LIN {X 0,Y 514.541,Z 472.109,A -85,B 0,C 180,E1 18530.323,E2 18530.323} C_VEL
LIN {X 0,Y 518.512,Z 477.461,A -85,B 0,C 180,E1 18528.318,E2 18528.318} C_VEL
LIN {X 0,Y 522.762,Z 483.32,A -85,B 0,C 180,E1 18526.449,E2 18526.449} C_VEL
LIN {X 0,Y 527.071,Z 489.295,A -85,B 0,C 180,E1 18524.767,E2 18524.767} C_VEL
LIN {X 0,Y 533.694,Z 498.743,A -85,B 0,C 180,E1 18522.472,E2 18522.472} C_VEL
LIN {X 0,Y 539.059,Z 506.974,A -85,B 0,C 180,E1 18520.795,E2 18520.795} C_VEL
LIN {X 0,Y 523.952,Z 728.007,A -85,B 0,C 180,E1 18517.35,E2 18517.35} C_VEL
LIN {X 0,Y 517.723,Z 820.272,A -85,B 0,C 180,E1 18515.894,E2 18515.894} C_VEL
LIN {X 0,Y 514.589,Z 848.021,A -85,B 0,C 180,E1 18515.355,E2 18515.355} C_VEL
LIN {X 0,Y 510.56,Z 873.327,A -85,B 0,C 180,E1 18514.692,E2 18514.692} C_VEL
LIN {X 0,Y 506.518,Z 894.443,A -85,B 0,C 180,E1 18514.008,E2 18514.008} C_VEL
LIN {X 0,Y 502.104,Z 914.553,A -85,B 0,C 180,E1 18513.226,E2 18513.226} C_VEL
LIN {X 0,Y 497.165,Z 934.488,A -85,B 0,C 180,E1 18512.317,E2 18512.317} C_VEL
LIN {X 0,Y 491.161,Z 956.295,A -85,B 0,C 180,E1 18511.152,E2 18511.152} C_VEL
LIN {X 0,Y 483.255,Z 981.832,A -85,B 0,C 180,E1 18509.524,E2 18509.524} C_VEL
LIN {X 0,Y 476.642,Z 1001.338,A -85,B 0,C 180,E1 18508.063,E2 18508.063} C_VEL
LIN {X 0,Y 470.058,Z 1019.621,A -85,B 0,C 180,E1 18506.493,E2 18506.493} C_VEL
LIN {X 0,Y 462.853,Z 1038.675,A -85,B 0,C 180,E1 18504.623,E2 18504.623} C_VEL
LIN {X 0,Y 453.945,Z 1061.048,A -85,B 0,C 180,E1 18502.048,E2 18502.048} C_VEL
LIN {X 0,Y 447.24,Z 1077.33,A -85,B 0,C 180,E1 18499.87,E2 18499.87} C_VEL
LIN {X 0,Y 441.126,Z 1092.029,A -85,B 0,C 180,E1 18497.639,E2 18497.639} C_VEL
LIN {X 0,Y 434.952,Z 1106.936,A -85,B 0,C 180,E1 18495.074,E2 18495.074} C_VEL
LIN {X 0,Y 427.824,Z 1124.354,A -85,B 0,C 180,E1 18491.585,E2 18491.585} C_VEL
LIN {X 0,Y 423.062,Z 1136.506,A -85,B 0,C 180,E1 18488.744,E2 18488.744} C_VEL
LIN {X 0,Y 419.152,Z 1147.094,A -85,B 0,C 180,E1 18485.931,E2 18485.931} C_VEL
LIN {X 0,Y 415.76,Z 1157.018,A -85,B 0,C 180,E1 18482.922,E2 18482.922} C_VEL
LIN {X 0,Y 412.455,Z 1168.021,A -85,B 0,C 180,E1 18479.001,E2 18479.001} C_VEL
LIN {X 0,Y 410.434,Z 1175.985,A -85,B 0,C 180,E1 18475.543,E2 18475.543} C_VEL
LIN {X 0,Y 409.286,Z 1181.753,A -85,B 0,C 180,E1 18472.553,E2 18472.553} C_VEL
LIN {X 0,Y 408.55,Z 1186.458,A -85,B 0,C 180,E1 18469.59,E2 18469.59} C_VEL
LIN {X 0,Y 408.161,Z 1190.139,A -85,B 0,C 180,E1 18466.655,E2 18466.655} C_VEL
LIN {X 0,Y 407.98,Z 1192.833,A -85,B 0,C 180,E1 18463.752,E2 18463.752} C_VEL
LIN {X 0,Y 407.922,Z 1194.569,A -85,B 0,C 180,E1 18460.879,E2 18460.879} C_VEL
LIN {X 0,Y 407.905,Z 1195.381,A -85,B 0,C 180,E1 18457.977,E2 18457.977} C_VEL
LIN {X 0,Y 407.916,Z 1195.427,A -85,B 0,C 180,E1 18456.222,E2 18456.222} C_VEL
LIN {X 0,Y 406.93,Z 1195.271,A -85,B 0,C 180,E1 18455.141,E2 18455.141} C_VEL
LIN {X 0,Y 402.464,Z 1194.759,A -85,B 0,C 180,E1 18453.178,E2 18453.178} C_VEL
LIN {X 0,Y 400.134,Z 1194.102,A -85,B 0,C 180,E1 18451.777,E2 18451.777} C_VEL
LIN {X 0,Y 399.947,Z 1193.873,A -85,B 0,C 180,E1 18451.298,E2 18451.298} C_VEL
LIN {X 0,Y 400.135,Z 1190.746,A -85,B 0,C 180,E1 18447.565,E2 18447.565} C_VEL
LIN {X 0,Y 400.536,Z 1186.971,A -85,B 0,C 180,E1 18444.413,E2 18444.413} C_VEL
LIN {X 0,Y 401.262,Z 1182.348,A -85,B 0,C 180,E1 18441.402,E2 18441.402} C_VEL
LIN {X 0,Y 402.426,Z 1176.694,A -85,B 0,C 180,E1 18438.39,E2 18438.39} C_VEL
LIN {X 0,Y 404.11,Z 1169.973,A -85,B 0,C 180,E1 18435.382,E2 18435.382} C_VEL
LIN {X 0,Y 406.636,Z 1161.349,A -85,B 0,C 180,E1 18432.1,E2 18432.1} C_VEL
LIN {X 0,Y 410.803,Z 1148.852,A -85,B 0,C 180,E1 18428.137,E2 18428.137} C_VEL
LIN {X 0,Y 414.762,Z 1137.944,A -85,B 0,C 180,E1 18425.2,E2 18425.2} C_VEL
LIN {X 0,Y 418.993,Z 1126.868,A -85,B 0,C 180,E1 18422.577,E2 18422.577} C_VEL
LIN {X 0,Y 423.994,Z 1114.24,A -85,B 0,C 180,E1 18419.939,E2 18419.939} C_VEL
LIN {X 0,Y 430.697,Z 1097.792,A -85,B 0,C 180,E1 18416.938,E2 18416.938} C_VEL
LIN {X 0,Y 437.793,Z 1079.937,A -85,B 0,C 180,E1 18414.174,E2 18414.174} C_VEL
LIN {X 0,Y 443.949,Z 1064.334,A -85,B 0,C 180,E1 18412.059,E2 18412.059} C_VEL
LIN {X 0,Y 450.043,Z 1048.496,A -85,B 0,C 180,E1 18410.159,E2 18410.159} C_VEL
LIN {X 0,Y 456.669,Z 1030.666,A -85,B 0,C 180,E1 18408.272,E2 18408.272} C_VEL
LIN {X 0,Y 465.037,Z 1006.737,A -85,B 0,C 180,E1 18406.101,E2 18406.101} C_VEL
LIN {X 0,Y 471.267,Z 987.54,A -85,B 0,C 180,E1 18404.611,E2 18404.611} C_VEL
LIN {X 0,Y 476.948,Z 968.674,A -85,B 0,C 180,E1 18403.328,E2 18403.328} C_VEL
LIN {X 0,Y 482.604,Z 948.292,A -85,B 0,C 180,E1 18402.124,E2 18402.124} C_VEL
LIN {X 0,Y 488.772,Z 923.824,A -85,B 0,C 180,E1 18400.892,E2 18400.892} C_VEL
LIN {X 0,Y 494.214,Z 898.257,A -85,B 0,C 180,E1 18399.846,E2 18399.846} C_VEL
LIN {X 0,Y 498.2,Z 876.459,A -85,B 0,C 180,E1 18399.111,E2 18399.111} C_VEL
LIN {X 0,Y 501.467,Z 855.255,A -85,B 0,C 180,E1 18398.525,E2 18398.525} C_VEL
LIN {X 0,Y 504.339,Z 832.162,A -85,B 0,C 180,E1 18398.02,E2 18398.02} C_VEL
LIN {X 0,Y 507.084,Z 796.287,A -85,B 0,C 180,E1 18397.415,E2 18397.415} C_VEL
LIN {X 0,Y 520.447,Z 572.17,A -85,B 0,C 180,E1 18393.945,E2 18393.945} C_VEL
LIN {X 0,Y 524.409,Z 506.936,A -85,B 0,C 180,E1 18392.916,E2 18392.916} C_VEL
LIN {X 0,Y 515.302,Z 493.27,A -85,B 0,C 180,E1 18390.589,E2 18390.589} C_VEL
LIN {X 0,Y 506.344,Z 480.4,A -85,B 0,C 180,E1 18388.033,E2 18388.033} C_VEL
LIN {X 0,Y 498.92,Z 470.251,A -85,B 0,C 180,E1 18385.651,E2 18385.651} C_VEL
LIN {X 0,Y 494.57,Z 464.457,A -85,B 0,C 180,E1 18384.104,E2 18384.104} C_VEL
LIN {X 0,Y 491.363,Z 460.243,A -85,B 0,C 180,E1 18382.872,E2 18382.872} C_VEL
LIN {X 0,Y 487.688,Z 455.452,A -85,B 0,C 180,E1 18381.341,E2 18381.341} C_VEL
LIN {X 0,Y 483.606,Z 450.143,A -85,B 0,C 180,E1 18379.444,E2 18379.444} C_VEL
LIN {X 0,Y 479.486,Z 444.918,A -85,B 0,C 180,E1 18377.244,E2 18377.244} C_VEL
LIN {X 0,Y 476.311,Z 441.329,A -85,B 0,C 180,E1 18375.275,E2 18375.275} C_VEL
LIN {X 0,Y 475.115,Z 439.249,A -85,B 0,C 180,E1 18374.379,E2 18374.379} C_VEL
LIN {X 0,Y 472.029,Z 436.36,A -85,B 0,C 180,E1 18371.857,E2 18371.857} C_VEL
LIN {X 0,Y 470.403,Z 433.167,A -85,B 0,C 180,E1 18369.914,E2 18369.914} C_VEL
LIN {X 0,Y 467.781,Z 431.545,A -85,B 0,C 180,E1 18364.045,E2 18364.045} C_VEL
LIN {X 0,Y 468.554,Z 432.213,A -85,B 0,C 180,E1 18360,E2 18360} C_VEL
LIN {X 0,Y 470.689,Z 433.52,A -85,B 0,C 180,E1 18356.834,E2 18356.834} C_VEL
LIN {X 0,Y 472.775,Z 437.369,A -85,B 0,C 180,E1 18354.539,E2 18354.539} C_VEL
LIN {X 0,Y 475.407,Z 439.641,A -85,B 0,C 180,E1 18352.507,E2 18352.507} C_VEL
LIN {X 0,Y 478.181,Z 443.702,A -85,B 0,C 180,E1 18350.613,E2 18350.613} C_VEL
LIN {X 0,Y 480.232,Z 445.708,A -85,B 0,C 180,E1 18349.442,E2 18349.442} C_VEL
LIN {X 0,Y 483.756,Z 450.314,A -85,B 0,C 180,E1 18347.587,E2 18347.587} C_VEL
LIN {X 0,Y 489.426,Z 457.654,A -85,B 0,C 180,E1 18345.023,E2 18345.023} C_VEL
LIN {X 0,Y 493.652,Z 463.214,A -85,B 0,C 180,E1 18343.345,E2 18343.345} C_VEL
LIN {X 0,Y 498.77,Z 470.057,A -85,B 0,C 180,E1 18341.503,E2 18341.503} C_VEL
LIN {X 0,Y 505.342,Z 478.953,A -85,B 0,C 180,E1 18339.378,E2 18339.378} C_VEL
LIN {X 0,Y 511.266,Z 487.935,A -85,B 0,C 180,E1 18337.612,E2 18337.612} C_VEL
LIN {X 0,Y 520.655,Z 502.964,A -85,B 0,C 180,E1 18335.068,E2 18335.068} C_VEL
LIN {X 0,Y 524.429,Z 509.627,A -85,B 0,C 180,E1 18334.109,E2 18334.109} C_VEL
LIN {X 0,Y 511.272,Z 727.01,A -85,B 0,C 180,E1 18330.736,E2 18330.736} C_VEL
LIN {X 0,Y 505.302,Z 825.794,A -85,B 0,C 180,E1 18329.189,E2 18329.189} C_VEL
LIN {X 0,Y 502.366,Z 853.611,A -85,B 0,C 180,E1 18328.652,E2 18328.652} C_VEL
LIN {X 0,Y 498.441,Z 879.544,A -85,B 0,C 180,E1 18327.977,E2 18327.977} C_VEL
LIN {X 0,Y 494.631,Z 900.61,A -85,B 0,C 180,E1 18327.295,E2 18327.295} C_VEL
LIN {X 0,Y 490.381,Z 921.029,A -85,B 0,C 180,E1 18326.504,E2 18326.504} C_VEL
LIN {X 0,Y 485.26,Z 942.822,A -85,B 0,C 180,E1 18325.505,E2 18325.505} C_VEL
LIN {X 0,Y 478.136,Z 969.65,A -85,B 0,C 180,E1 18324.025,E2 18324.025} C_VEL
LIN {X 0,Y 472.04,Z 990.095,A -85,B 0,C 180,E1 18322.69,E2 18322.69} C_VEL
LIN {X 0,Y 466.19,Z 1008.36,A -85,B 0,C 180,E1 18321.323,E2 18321.323} C_VEL
LIN {X 0,Y 460.135,Z 1026.2,A -85,B 0,C 180,E1 18319.805,E2 18319.805} C_VEL
LIN {X 0,Y 453.465,Z 1044.906,A -85,B 0,C 180,E1 18317.993,E2 18317.993} C_VEL
LIN {X 0,Y 444.933,Z 1067.602,A -85,B 0,C 180,E1 18315.428,E2 18315.428} C_VEL
LIN {X 0,Y 438.299,Z 1084.613,A -85,B 0,C 180,E1 18313.186,E2 18313.186} C_VEL
LIN {X 0,Y 432.59,Z 1099.07,A -85,B 0,C 180,E1 18311.027,E2 18311.027} C_VEL
LIN {X 0,Y 426.774,Z 1113.76,A -85,B 0,C 180,E1 18308.549,E2 18308.549} C_VEL
LIN {X 0,Y 420.3,Z 1130.399,A -85,B 0,C 180,E1 18305.314,E2 18305.314} C_VEL
LIN {X 0,Y 415.223,Z 1143.634,A -85,B 0,C 180,E1 18302.302,E2 18302.302} C_VEL
LIN {X 0,Y 411.387,Z 1154.324,A -85,B 0,C 180,E1 18299.526,E2 18299.526} C_VEL
LIN {X 0,Y 408.025,Z 1164.334,A -85,B 0,C 180,E1 18296.561,E2 18296.561} C_VEL
LIN {X 0,Y 405.122,Z 1173.984,A -85,B 0,C 180,E1 18293.259,E2 18293.259} C_VEL
LIN {X 0,Y 402.652,Z 1183.587,A -85,B 0,C 180,E1 18289.285,E2 18289.285} C_VEL
LIN {X 0,Y 401.344,Z 1189.964,A -85,B 0,C 180,E1 18286.053,E2 18286.053} C_VEL
LIN {X 0,Y 400.584,Z 1194.712,A -85,B 0,C 180,E1 18283.128,E2 18283.128} C_VEL
LIN {X 0,Y 400.164,Z 1198.608,A -85,B 0,C 180,E1 18280.103,E2 18280.103} C_VEL
LIN {X 0,Y 399.99,Z 1201.293,A -85,B 0,C 180,E1 18277.324,E2 18277.324} C_VEL
LIN {X 0,Y 399.919,Z 1203.173,A -85,B 0,C 180,E1 18274.445,E2 18274.445} C_VEL
LIN {X 0,Y 399.91,Z 1204.11,A -85,B 0,C 180,E1 18271.719,E2 18271.719} C_VEL
LIN {X 0,Y 399.913,Z 1204.201,A -85,B 0,C 180,E1 18268.854,E2 18268.854} C_VEL
LIN {X 0,Y 399.916,Z 1203.377,A -85,B 0,C 180,E1 18265.986,E2 18265.986} C_VEL
LIN {X 0,Y 399.967,Z 1201.638,A -85,B 0,C 180,E1 18263.108,E2 18263.108} C_VEL
LIN {X 0,Y 400.134,Z 1198.975,A -85,B 0,C 180,E1 18260.217,E2 18260.217} C_VEL
LIN {X 0,Y 400.528,Z 1195.167,A -85,B 0,C 180,E1 18257.163,E2 18257.163} C_VEL
LIN {X 0,Y 401.256,Z 1190.564,A -85,B 0,C 180,E1 18254.24,E2 18254.24} C_VEL
LIN {X 0,Y 402.439,Z 1184.673,A -85,B 0,C 180,E1 18251.157,E2 18251.157} C_VEL
LIN {X 0,Y 404.211,Z 1177.671,A -85,B 0,C 180,E1 18248.068,E2 18248.068} C_VEL
LIN {X 0,Y 407.314,Z 1167.466,A -85,B 0,C 180,E1 18244.247,E2 18244.247} C_VEL
LIN {X 0,Y 411.361,Z 1155.632,A -85,B 0,C 180,E1 18240.595,E2 18240.595} C_VEL
LIN {X 0,Y 415.406,Z 1144.863,A -85,B 0,C 180,E1 18237.701,E2 18237.701} C_VEL
LIN {X 0,Y 420.273,Z 1132.771,A -85,B 0,C 180,E1 18234.849,E2 18234.849} C_VEL
LIN {X 0,Y 426.871,Z 1117.144,A -85,B 0,C 180,E1 18231.632,E2 18231.632} C_VEL
LIN {X 0,Y 434.143,Z 1099.904,A -85,B 0,C 180,E1 18228.626,E2 18228.626} C_VEL
LIN {X 0,Y 440.46,Z 1085.089,A -85,B 0,C 180,E1 18226.363,E2 18226.363} C_VEL
LIN {X 0,Y 447.076,Z 1069.432,A -85,B 0,C 180,E1 18224.25,E2 18224.25} C_VEL
LIN {X 0,Y 455.489,Z 1049.155,A -85,B 0,C 180,E1 18221.862,E2 18221.862} C_VEL
LIN {X 0,Y 463.944,Z 1027.412,A -85,B 0,C 180,E1 18219.702,E2 18219.702} C_VEL
LIN {X 0,Y 470.794,Z 1008.909,A -85,B 0,C 180,E1 18218.107,E2 18218.107} C_VEL
LIN {X 0,Y 477.681,Z 989.169,A -85,B 0,C 180,E1 18216.625,E2 18216.625} C_VEL
LIN {X 0,Y 485.495,Z 965.019,A -85,B 0,C 180,E1 18215.072,E2 18215.072} C_VEL
LIN {X 0,Y 492.199,Z 941.436,A -85,B 0,C 180,E1 18213.814,E2 18213.814} C_VEL
LIN {X 0,Y 497.27,Z 921.68,A -85,B 0,C 180,E1 18212.917,E2 18212.917} C_VEL
LIN {X 0,Y 501.906,Z 901.407,A -85,B 0,C 180,E1 18212.135,E2 18212.135} C_VEL
LIN {X 0,Y 506.047,Z 880.54,A -85,B 0,C 180,E1 18211.461,E2 18211.461} C_VEL
LIN {X 0,Y 509.796,Z 858.126,A -85,B 0,C 180,E1 18210.873,E2 18210.873} C_VEL
LIN {X 0,Y 513.507,Z 828.706,A -85,B 0,C 180,E1 18210.283,E2 18210.283} C_VEL
LIN {X 0,Y 517.306,Z 776.027,A -85,B 0,C 180,E1 18209.44,E2 18209.44} C_VEL
LIN {X 0,Y 532.526,Z 555.952,A -85,B 0,C 180,E1 18206.005,E2 18206.005} C_VEL
LIN {X 0,Y 535.526,Z 513.871,A -85,B 0,C 180,E1 18205.34,E2 18205.34} C_VEL
LIN {X 0,Y 530.021,Z 504.697,A -85,B 0,C 180,E1 18203.516,E2 18203.516} C_VEL
LIN {X 0,Y 523.348,Z 494.052,A -85,B 0,C 180,E1 18201.021,E2 18201.021} C_VEL
LIN {X 0,Y 518.979,Z 487.856,A -85,B 0,C 180,E1 18199.177,E2 18199.177} C_VEL
LIN {X 0,Y 515.666,Z 483.285,A -85,B 0,C 180,E1 18197.607,E2 18197.607} C_VEL
LIN {X 0,Y 512.04,Z 478.241,A -85,B 0,C 180,E1 18195.633,E2 18195.633} C_VEL
LIN {X 0,Y 508.794,Z 473.79,A -85,B 0,C 180,E1 18193.525,E2 18193.525} C_VEL
LIN {X 0,Y 504.983,Z 468.841,A -85,B 0,C 180,E1 18190.247,E2 18190.247} C_VEL
LIN {X 0,Y 504.344,Z 467.593,A -85,B 0,C 180,E1 18189.471,E2 18189.471} C_VEL
LIN {X 0,Y 501.757,Z 465.408,A -85,B 0,C 180,E1 18184.114,E2 18184.114} C_VEL
LIN {X 0,Y 502.105,Z 465.864,A -85,B 0,C 180,E1 18181.027,E2 18181.027} C_VEL
LIN {X 0,Y 504.615,Z 467.919,A -85,B 0,C 180,E1 18177.007,E2 18177.007} C_VEL
LIN {X 0,Y 507.047,Z 472.025,A -85,B 0,C 180,E1 18174.568,E2 18174.568} C_VEL
LIN {X 0,Y 508.847,Z 473.888,A -85,B 0,C 180,E1 18173.229,E2 18173.229} C_VEL
LIN {X 0,Y 512.1,Z 478.311,A -85,B 0,C 180,E1 18171.127,E2 18171.127} C_VEL
LIN {X 0,Y 517.051,Z 485.162,A -85,B 0,C 180,E1 18168.511,E2 18168.511} C_VEL
LIN {X 0,Y 521.242,Z 491.03,A -85,B 0,C 180,E1 18166.635,E2 18166.635} C_VEL
LIN {X 0,Y 526.846,Z 498.837,A -85,B 0,C 180,E1 18164.45,E2 18164.45} C_VEL
LIN {X 0,Y 533.524,Z 508.845,A -85,B 0,C 180,E1 18162.156,E2 18162.156} C_VEL
LIN {X 0,Y 535.563,Z 512.091,A -85,B 0,C 180,E1 18161.506,E2 18161.506} C_VEL
LIN {X 0,Y 520.129,Z 731.771,A -85,B 0,C 180,E1 18158.081,E2 18158.081} C_VEL
LIN {X 0,Y 513.954,Z 820.365,A -85,B 0,C 180,E1 18156.681,E2 18156.681} C_VEL
LIN {X 0,Y 510.733,Z 848.221,A -85,B 0,C 180,E1 18156.141,E2 18156.141} C_VEL
LIN {X 0,Y 506.612,Z 873.503,A -85,B 0,C 180,E1 18155.482,E2 18155.482} C_VEL
LIN {X 0,Y 502.423,Z 894.86,A -85,B 0,C 180,E1 18154.793,E2 18154.793} C_VEL
LIN {X 0,Y 497.816,Z 915.254,A -85,B 0,C 180,E1 18154,E2 18154} C_VEL
LIN {X 0,Y 492.459,Z 936.22,A -85,B 0,C 180,E1 18153.039,E2 18153.039} C_VEL
LIN {X 0,Y 485.143,Z 961.704,A -85,B 0,C 180,E1 18151.645,E2 18151.645} C_VEL
LIN {X 0,Y 478.062,Z 983.47,A -85,B 0,C 180,E1 18150.223,E2 18150.223} C_VEL
LIN {X 0,Y 471.582,Z 1001.971,A -85,B 0,C 180,E1 18148.827,E2 18148.827} C_VEL
LIN {X 0,Y 464.808,Z 1020.203,A -85,B 0,C 180,E1 18147.255,E2 18147.255} C_VEL
LIN {X 0,Y 457.273,Z 1039.458,A -85,B 0,C 180,E1 18145.352,E2 18145.352} C_VEL
LIN {X 0,Y 448.172,Z 1061.456,A -85,B 0,C 180,E1 18142.799,E2 18142.799} C_VEL
LIN {X 0,Y 441.208,Z 1077.72,A -85,B 0,C 180,E1 18140.603,E2 18140.603} C_VEL
LIN {X 0,Y 434.858,Z 1092.389,A -85,B 0,C 180,E1 18138.354,E2 18138.354} C_VEL
LIN {X 0,Y 428.096,Z 1108.054,A -85,B 0,C 180,E1 18135.618,E2 18135.618} C_VEL
LIN {X 0,Y 420.991,Z 1124.623,A -85,B 0,C 180,E1 18132.231,E2 18132.231} C_VEL
LIN {X 0,Y 416.03,Z 1136.639,A -85,B 0,C 180,E1 18129.381,E2 18129.381} C_VEL
LIN {X 0,Y 411.869,Z 1147.312,A -85,B 0,C 180,E1 18126.496,E2 18126.496} C_VEL
LIN {X 0,Y 408.214,Z 1157.454,A -85,B 0,C 180,E1 18123.357,E2 18123.357} C_VEL
LIN {X 0,Y 404.669,Z 1168.563,A -85,B 0,C 180,E1 18119.281,E2 18119.281} C_VEL
LIN {X 0,Y 402.627,Z 1176.129,A -85,B 0,C 180,E1 18115.917,E2 18115.917} C_VEL
LIN {X 0,Y 401.384,Z 1181.959,A -85,B 0,C 180,E1 18112.822,E2 18112.822} C_VEL
LIN {X 0,Y 400.592,Z 1186.665,A -85,B 0,C 180,E1 18109.778,E2 18109.778} C_VEL
LIN {X 0,Y 400.17,Z 1190.408,A -85,B 0,C 180,E1 18106.699,E2 18106.699} C_VEL
LIN {X 0,Y 399.972,Z 1193.25,A -85,B 0,C 180,E1 18103.476,E2 18103.476} C_VEL
LIN {X 0,Y 399.919,Z 1195.192,A -85,B 0,C 180,E1 18099.788,E2 18099.788} C_VEL
LIN {X 0,Y 399.917,Z 1195.507,A -85,B 0,C 180,E1 18096.172,E2 18096.172} C_VEL
LIN {X 0,Y 399.921,Z 1194.742,A -85,B 0,C 180,E1 18093.153,E2 18093.153} C_VEL
LIN {X 0,Y 399.947,Z 1193.873,A -85,B 0,C 180,E1 18091.298,E2 18091.298} C_VEL
LIN {X 0,Y 398.997,Z 1193.239,A -85,B 0,C 180,E1 18090.198,E2 18090.198} C_VEL
LIN {X 0,Y 392.716,Z 1190.512,A -85,B 0,C 180,E1 18087.106,E2 18087.106} C_VEL
LIN {X 0,Y 392.26,Z 1189.666,A -85,B 0,C 180,E1 18086.302,E2 18086.302} C_VEL
LIN {X 0,Y 392.921,Z 1185.006,A -85,B 0,C 180,E1 18082.69,E2 18082.69} C_VEL
LIN {X 0,Y 394.336,Z 1177.904,A -85,B 0,C 180,E1 18078.593,E2 18078.593} C_VEL
LIN {X 0,Y 396.111,Z 1171.018,A -85,B 0,C 180,E1 18075.379,E2 18075.379} C_VEL
LIN {X 0,Y 398.426,Z 1163.313,A -85,B 0,C 180,E1 18072.323,E2 18072.323} C_VEL
LIN {X 0,Y 401.433,Z 1154.436,A -85,B 0,C 180,E1 18069.287,E2 18069.287} C_VEL
LIN {X 0,Y 406.061,Z 1142.105,A -85,B 0,C 180,E1 18065.657,E2 18065.657} C_VEL
LIN {X 0,Y 411.325,Z 1128.633,A -85,B 0,C 180,E1 18062.336,E2 18062.336} C_VEL
LIN {X 0,Y 416.314,Z 1116.454,A -85,B 0,C 180,E1 18059.712,E2 18059.712} C_VEL
LIN {X 0,Y 421.667,Z 1103.641,A -85,B 0,C 180,E1 18057.273,E2 18057.273} C_VEL
LIN {X 0,Y 427.606,Z 1089.446,A -85,B 0,C 180,E1 18054.886,E2 18054.886} C_VEL
LIN {X 0,Y 435.503,Z 1070.486,A -85,B 0,C 180,E1 18052.11,E2 18052.11} C_VEL
LIN {X 0,Y 442.917,Z 1051.844,A -85,B 0,C 180,E1 18049.788,E2 18049.788} C_VEL
LIN {X 0,Y 449.374,Z 1035.064,A -85,B 0,C 180,E1 18047.954,E2 18047.954} C_VEL
LIN {X 0,Y 455.747,Z 1017.743,A -85,B 0,C 180,E1 18046.285,E2 18046.285} C_VEL
LIN {X 0,Y 462.6,Z 998.079,A -85,B 0,C 180,E1 18044.626,E2 18044.626} C_VEL
LIN {X 0,Y 470.773,Z 972.483,A -85,B 0,C 180,E1 18042.795,E2 18042.795} C_VEL
LIN {X 0,Y 476.812,Z 951.552,A -85,B 0,C 180,E1 18041.53,E2 18041.53} C_VEL
LIN {X 0,Y 481.99,Z 931.83,A -85,B 0,C 180,E1 18040.502,E2 18040.502} C_VEL
LIN {X 0,Y 486.964,Z 910.669,A -85,B 0,C 180,E1 18039.557,E2 18039.557} C_VEL
LIN {X 0,Y 492.453,Z 883.629,A -85,B 0,C 180,E1 18038.561,E2 18038.561} C_VEL
LIN {X 0,Y 496.502,Z 858.808,A -85,B 0,C 180,E1 18037.846,E2 18037.846} C_VEL
LIN {X 0,Y 499.366,Z 837.111,A -85,B 0,C 180,E1 18037.352,E2 18037.352} C_VEL
LIN {X 0,Y 501.535,Z 814.579,A -85,B 0,C 180,E1 18036.942,E2 18036.942} C_VEL
LIN {X 0,Y 514.745,Z 600.28,A -85,B 0,C 180,E1 18033.606,E2 18033.606} C_VEL
LIN {X 0,Y 520.293,Z 511.555,A -85,B 0,C 180,E1 18032.21,E2 18032.21} C_VEL
LIN {X 0,Y 510.446,Z 496.68,A -85,B 0,C 180,E1 18029.58,E2 18029.58} C_VEL
LIN {X 0,Y 501.167,Z 483.294,A -85,B 0,C 180,E1 18026.769,E2 18026.769} C_VEL
LIN {X 0,Y 493.611,Z 472.979,A -85,B 0,C 180,E1 18024.154,E2 18024.154} C_VEL
LIN {X 0,Y 489.413,Z 467.465,A -85,B 0,C 180,E1 18022.524,E2 18022.524} C_VEL
LIN {X 0,Y 486.073,Z 463.017,A -85,B 0,C 180,E1 18021.1,E2 18021.1} C_VEL
LIN {X 0,Y 482.054,Z 457.73,A -85,B 0,C 180,E1 18019.194,E2 18019.194} C_VEL
LIN {X 0,Y 478.292,Z 452.785,A -85,B 0,C 180,E1 18017.144,E2 18017.144} C_VEL
LIN {X 0,Y 474.998,Z 449.034,A -85,B 0,C 180,E1 18015.069,E2 18015.069} C_VEL
LIN {X 0,Y 473.819,Z 447.031,A -85,B 0,C 180,E1 18014.17,E2 18014.17} C_VEL
LIN {X 0,Y 470.817,Z 444.076,A -85,B 0,C 180,E1 18011.64,E2 18011.64} C_VEL
LIN {X 0,Y 469.334,Z 441.079,A -85,B 0,C 180,E1 18009.813,E2 18009.813} C_VEL
LIN {X 0,Y 466.805,Z 439.485,A -85,B 0,C 180,E1 18004.053,E2 18004.053} C_VEL
LIN {X 0,Y 467.576,Z 440.157,A -85,B 0,C 180,E1 18000,E2 18000} C_VEL
LIN {X 0,Y 469.601,Z 441.436,A -85,B 0,C 180,E1 17996.949,E2 17996.949} C_VEL
LIN {X 0,Y 471.656,Z 445.241,A -85,B 0,C 180,E1 17994.648,E2 17994.648} C_VEL
LIN {X 0,Y 474.169,Z 447.478,A -85,B 0,C 180,E1 17992.67,E2 17992.67} C_VEL
LIN {X 0,Y 477.003,Z 451.586,A -85,B 0,C 180,E1 17990.711,E2 17990.711} C_VEL
LIN {X 0,Y 478.824,Z 453.407,A -85,B 0,C 180,E1 17989.654,E2 17989.654} C_VEL
LIN {X 0,Y 482.414,Z 458.106,A -85,B 0,C 180,E1 17987.734,E2 17987.734} C_VEL
LIN {X 0,Y 487.885,Z 465.381,A -85,B 0,C 180,E1 17985.217,E2 17985.217} C_VEL
LIN {X 0,Y 491.989,Z 470.863,A -85,B 0,C 180,E1 17983.56,E2 17983.56} C_VEL
LIN {X 0,Y 498.576,Z 479.657,A -85,B 0,C 180,E1 17981.193,E2 17981.193} C_VEL
LIN {X 0,Y 505.797,Z 489.962,A -85,B 0,C 180,E1 17978.882,E2 17978.882} C_VEL
LIN {X 0,Y 516.299,Z 506.899,A -85,B 0,C 180,E1 17975.881,E2 17975.881} C_VEL
LIN {X 0,Y 520.334,Z 513.973,A -85,B 0,C 180,E1 17974.816,E2 17974.816} C_VEL
LIN {X 0,Y 506.749,Z 732.106,A -85,B 0,C 180,E1 17971.427,E2 17971.427} C_VEL
LIN {X 0,Y 500.917,Z 825.772,A -85,B 0,C 180,E1 17969.955,E2 17969.955} C_VEL
LIN {X 0,Y 497.915,Z 853.564,A -85,B 0,C 180,E1 17969.418,E2 17969.418} C_VEL
LIN {X 0,Y 493.894,Z 879.509,A -85,B 0,C 180,E1 17968.745,E2 17968.745} C_VEL
LIN {X 0,Y 489.912,Z 900.999,A -85,B 0,C 180,E1 17968.049,E2 17968.049} C_VEL
LIN {X 0,Y 485.428,Z 921.952,A -85,B 0,C 180,E1 17967.234,E2 17967.234} C_VEL
LIN {X 0,Y 479.761,Z 945.371,A -85,B 0,C 180,E1 17966.15,E2 17966.15} C_VEL
LIN {X 0,Y 472.742,Z 970.746,A -85,B 0,C 180,E1 17964.725,E2 17964.725} C_VEL
LIN {X 0,Y 466.758,Z 990.243,A -85,B 0,C 180,E1 17963.446,E2 17963.446} C_VEL
LIN {X 0,Y 460.495,Z 1009.248,A -85,B 0,C 180,E1 17962.015,E2 17962.015} C_VEL
LIN {X 0,Y 454.024,Z 1027.724,A -85,B 0,C 180,E1 17960.423,E2 17960.423} C_VEL
LIN {X 0,Y 445.921,Z 1049.671,A -85,B 0,C 180,E1 17958.243,E2 17958.243} C_VEL
LIN {X 0,Y 438.21,Z 1069.244,A -85,B 0,C 180,E1 17955.95,E2 17955.95} C_VEL
LIN {X 0,Y 431.785,Z 1085.159,A -85,B 0,C 180,E1 17953.818,E2 17953.818} C_VEL
LIN {X 0,Y 425.54,Z 1100.435,A -85,B 0,C 180,E1 17951.498,E2 17951.498} C_VEL
LIN {X 0,Y 418.65,Z 1117.355,A -85,B 0,C 180,E1 17948.561,E2 17948.561} C_VEL
LIN {X 0,Y 412.34,Z 1132.708,A -85,B 0,C 180,E1 17945.418,E2 17945.418} C_VEL
LIN {X 0,Y 407.673,Z 1144.503,A -85,B 0,C 180,E1 17942.654,E2 17942.654} C_VEL
LIN {X 0,Y 403.742,Z 1155.023,A -85,B 0,C 180,E1 17939.853,E2 17939.853} C_VEL
LIN {X 0,Y 400.163,Z 1165.286,A -85,B 0,C 180,E1 17936.728,E2 17936.728} C_VEL
LIN {X 0,Y 396.693,Z 1176.5,A -85,B 0,C 180,E1 17932.683,E2 17932.683} C_VEL
LIN {X 0,Y 394.693,Z 1184.054,A -85,B 0,C 180,E1 17929.381,E2 17929.381} C_VEL
LIN {X 0,Y 393.4,Z 1190.089,A -85,B 0,C 180,E1 17926.235,E2 17926.235} C_VEL
LIN {X 0,Y 392.608,Z 1194.802,A -85,B 0,C 180,E1 17923.25,E2 17923.25} C_VEL
LIN {X 0,Y 392.174,Z 1198.605,A -85,B 0,C 180,E1 17920.214,E2 17920.214} C_VEL
LIN {X 0,Y 391.989,Z 1201.307,A -85,B 0,C 180,E1 17917.327,E2 17917.327} C_VEL
LIN {X 0,Y 391.92,Z 1203.078,A -85,B 0,C 180,E1 17914.536,E2 17914.536} C_VEL
LIN {X 0,Y 391.91,Z 1204.02,A -85,B 0,C 180,E1 17911.754,E2 17911.754} C_VEL
LIN {X 0,Y 391.914,Z 1204.115,A -85,B 0,C 180,E1 17908.831,E2 17908.831} C_VEL
LIN {X 0,Y 391.916,Z 1203.296,A -85,B 0,C 180,E1 17905.904,E2 17905.904} C_VEL
LIN {X 0,Y 391.976,Z 1201.5,A -85,B 0,C 180,E1 17902.887,E2 17902.887} C_VEL
LIN {X 0,Y 392.167,Z 1198.746,A -85,B 0,C 180,E1 17899.868,E2 17899.868} C_VEL
LIN {X 0,Y 392.579,Z 1195.11,A -85,B 0,C 180,E1 17896.899,E2 17896.899} C_VEL
LIN {X 0,Y 393.361,Z 1190.517,A -85,B 0,C 180,E1 17893.914,E2 17893.914} C_VEL
LIN {X 0,Y 394.633,Z 1184.643,A -85,B 0,C 180,E1 17890.769,E2 17890.769} C_VEL
LIN {X 0,Y 396.521,Z 1177.657,A -85,B 0,C 180,E1 17887.619,E2 17887.619} C_VEL
LIN {X 0,Y 399.807,Z 1167.483,A -85,B 0,C 180,E1 17883.727,E2 17883.727} C_VEL
LIN {X 0,Y 404.078,Z 1155.665,A -85,B 0,C 180,E1 17880.006,E2 17880.006} C_VEL
LIN {X 0,Y 408.343,Z 1144.933,A -85,B 0,C 180,E1 17877.072,E2 17877.072} C_VEL
LIN {X 0,Y 413.176,Z 1133.5,A -85,B 0,C 180,E1 17874.324,E2 17874.324} C_VEL
LIN {X 0,Y 419.791,Z 1118.462,A -85,B 0,C 180,E1 17871.158,E2 17871.158} C_VEL
LIN {X 0,Y 427.549,Z 1100.922,A -85,B 0,C 180,E1 17868.023,E2 17868.023} C_VEL
LIN {X 0,Y 434.479,Z 1085.311,A -85,B 0,C 180,E1 17865.606,E2 17865.606} C_VEL
LIN {X 0,Y 441.409,Z 1069.516,A -85,B 0,C 180,E1 17863.458,E2 17863.458} C_VEL
LIN {X 0,Y 450.068,Z 1049.385,A -85,B 0,C 180,E1 17861.074,E2 17861.074} C_VEL
LIN {X 0,Y 458.765,Z 1027.793,A -85,B 0,C 180,E1 17858.916,E2 17858.916} C_VEL
LIN {X 0,Y 465.815,Z 1009.353,A -85,B 0,C 180,E1 17857.32,E2 17857.32} C_VEL
LIN {X 0,Y 472.754,Z 990.059,A -85,B 0,C 180,E1 17855.864,E2 17855.864} C_VEL
LIN {X 0,Y 480.094,Z 968.131,A -85,B 0,C 180,E1 17854.44,E2 17854.44} C_VEL
LIN {X 0,Y 487.792,Z 942.188,A -85,B 0,C 180,E1 17853.034,E2 17853.034} C_VEL
LIN {X 0,Y 493.396,Z 920.871,A -85,B 0,C 180,E1 17852.07,E2 17852.07} C_VEL
LIN {X 0,Y 498.158,Z 900.449,A -85,B 0,C 180,E1 17851.293,E2 17851.293} C_VEL
LIN {X 0,Y 502.445,Z 879.192,A -85,B 0,C 180,E1 17850.616,E2 17850.616} C_VEL
LIN {X 0,Y 506.831,Z 853.258,A -85,B 0,C 180,E1 17849.958,E2 17849.958} C_VEL
LIN {X 0,Y 510.116,Z 825.477,A -85,B 0,C 180,E1 17849.429,E2 17849.429} C_VEL
LIN {X 0,Y 517.254,Z 725.256,A -85,B 0,C 180,E1 17847.847,E2 17847.847} C_VEL
LIN {X 0,Y 532.153,Z 518.787,A -85,B 0,C 180,E1 17844.624,E2 17844.624} C_VEL
LIN {X 0,Y 524.714,Z 506.488,A -85,B 0,C 180,E1 17841.99,E2 17841.99} C_VEL
LIN {X 0,Y 520.347,Z 499.65,A -85,B 0,C 180,E1 17840.236,E2 17840.236} C_VEL
LIN {X 0,Y 516.932,Z 494.804,A -85,B 0,C 180,E1 17838.729,E2 17838.729} C_VEL
LIN {X 0,Y 514.042,Z 490.737,A -85,B 0,C 180,E1 17837.314,E2 17837.314} C_VEL
LIN {X 0,Y 510.694,Z 485.955,A -85,B 0,C 180,E1 17835.443,E2 17835.443} C_VEL
LIN {X 0,Y 507.513,Z 481.496,A -85,B 0,C 180,E1 17833.327,E2 17833.327} C_VEL
LIN {X 0,Y 503.822,Z 476.579,A -85,B 0,C 180,E1 17830.058,E2 17830.058} C_VEL
LIN {X 0,Y 503.275,Z 475.497,A -85,B 0,C 180,E1 17829.376,E2 17829.376} C_VEL
LIN {X 0,Y 500.771,Z 473.331,A -85,B 0,C 180,E1 17824.007,E2 17824.007} C_VEL
LIN {X 0,Y 501.163,Z 473.862,A -85,B 0,C 180,E1 17820.915,E2 17820.915} C_VEL
LIN {X 0,Y 503.499,Z 475.749,A -85,B 0,C 180,E1 17817.154,E2 17817.154} C_VEL
LIN {X 0,Y 506.062,Z 480.048,A -85,B 0,C 180,E1 17814.558,E2 17814.558} C_VEL
LIN {X 0,Y 507.621,Z 481.704,A -85,B 0,C 180,E1 17813.383,E2 17813.383} C_VEL
LIN {X 0,Y 510.922,Z 486.191,A -85,B 0,C 180,E1 17811.22,E2 17811.22} C_VEL
LIN {X 0,Y 515.597,Z 492.859,A -85,B 0,C 180,E1 17808.704,E2 17808.704} C_VEL
LIN {X 0,Y 519.604,Z 498.553,A -85,B 0,C 180,E1 17806.875,E2 17806.875} C_VEL
LIN {X 0,Y 524.981,Z 506.177,A -85,B 0,C 180,E1 17804.733,E2 17804.733} C_VEL
LIN {X 0,Y 531.55,Z 516.198,A -85,B 0,C 180,E1 17802.427,E2 17802.427} C_VEL
LIN {X 0,Y 532.146,Z 517.318,A -85,B 0,C 180,E1 17802.225,E2 17802.225} C_VEL
LIN {X 0,Y 516.403,Z 735.346,A -85,B 0,C 180,E1 17798.826,E2 17798.826} C_VEL
LIN {X 0,Y 510.276,Z 820.692,A -85,B 0,C 180,E1 17797.476,E2 17797.476} C_VEL
LIN {X 0,Y 506.932,Z 848.728,A -85,B 0,C 180,E1 17796.933,E2 17796.933} C_VEL
LIN {X 0,Y 502.763,Z 873.691,A -85,B 0,C 180,E1 17796.285,E2 17796.285} C_VEL
LIN {X 0,Y 498.633,Z 894.312,A -85,B 0,C 180,E1 17795.624,E2 17795.624} C_VEL
LIN {X 0,Y 493.842,Z 915.065,A -85,B 0,C 180,E1 17794.826,E2 17794.826} C_VEL
LIN {X 0,Y 488.471,Z 935.626,A -85,B 0,C 180,E1 17793.89,E2 17793.89} C_VEL
LIN {X 0,Y 481.459,Z 959.677,A -85,B 0,C 180,E1 17792.598,E2 17792.598} C_VEL
LIN {X 0,Y 473.589,Z 983.262,A -85,B 0,C 180,E1 17791.07,E2 17791.07} C_VEL
LIN {X 0,Y 466.701,Z 1002.388,A -85,B 0,C 180,E1 17789.627,E2 17789.627} C_VEL
LIN {X 0,Y 459.644,Z 1020.788,A -85,B 0,C 180,E1 17788.034,E2 17788.034} C_VEL
LIN {X 0,Y 451.254,Z 1041.555,A -85,B 0,C 180,E1 17785.963,E2 17785.963} C_VEL
LIN {X 0,Y 442.317,Z 1062.237,A -85,B 0,C 180,E1 17783.521,E2 17783.521} C_VEL
LIN {X 0,Y 435.258,Z 1078.127,A -85,B 0,C 180,E1 17781.355,E2 17781.355} C_VEL
LIN {X 0,Y 428.496,Z 1093.135,A -85,B 0,C 180,E1 17779.026,E2 17779.026} C_VEL
LIN {X 0,Y 420.947,Z 1109.985,A -85,B 0,C 180,E1 17776.03,E2 17776.03} C_VEL
LIN {X 0,Y 413.91,Z 1125.575,A -85,B 0,C 180,E1 17772.745,E2 17772.745} C_VEL
LIN {X 0,Y 408.756,Z 1137.483,A -85,B 0,C 180,E1 17769.857,E2 17769.857} C_VEL
LIN {X 0,Y 404.422,Z 1148.073,A -85,B 0,C 180,E1 17766.925,E2 17766.925} C_VEL
LIN {X 0,Y 399.992,Z 1159.927,A -85,B 0,C 180,E1 17763.13,E2 17763.13} C_VEL
LIN {X 0,Y 396.683,Z 1169.767,A -85,B 0,C 180,E1 17759.291,E2 17759.291} C_VEL
LIN {X 0,Y 394.758,Z 1176.594,A -85,B 0,C 180,E1 17756.149,E2 17756.149} C_VEL
LIN {X 0,Y 393.466,Z 1182.282,A -85,B 0,C 180,E1 17753.038,E2 17753.038} C_VEL
LIN {X 0,Y 392.631,Z 1186.911,A -85,B 0,C 180,E1 17749.952,E2 17749.952} C_VEL
LIN {X 0,Y 392.18,Z 1190.684,A -85,B 0,C 180,E1 17746.744,E2 17746.744} C_VEL
LIN {X 0,Y 391.964,Z 1193.724,A -85,B 0,C 180,E1 17743.122,E2 17743.122} C_VEL
LIN {X 0,Y 391.916,Z 1195.35,A -85,B 0,C 180,E1 17739.397,E2 17739.397} C_VEL
LIN {X 0,Y 391.917,Z 1195.592,A -85,B 0,C 180,E1 17736.151,E2 17736.151} C_VEL
LIN {X 0,Y 391.923,Z 1194.82,A -85,B 0,C 180,E1 17733.071,E2 17733.071} C_VEL
LIN {X 0,Y 391.996,Z 1193.069,A -85,B 0,C 180,E1 17730,E2 17730} C_VEL
LIN {X 0,Y 392.196,Z 1190.339,A -85,B 0,C 180,E1 17726.931,E2 17726.931} C_VEL
LIN {X 0,Y 392.26,Z 1189.666,A -85,B 0,C 180,E1 17726.302,E2 17726.302} C_VEL
LIN {X 0,Y 391.408,Z 1188.503,A -85,B 0,C 180,E1 17725.188,E2 17725.188} C_VEL
LIN {X 0,Y 385.611,Z 1184.551,A -85,B 0,C 180,E1 17722.048,E2 17722.048} C_VEL
LIN {X 0,Y 385.324,Z 1183.25,A -85,B 0,C 180,E1 17721.242,E2 17721.242} C_VEL
LIN {X 0,Y 386.667,Z 1177.336,A -85,B 0,C 180,E1 17717.91,E2 17717.91} C_VEL
LIN {X 0,Y 388.518,Z 1170.68,A -85,B 0,C 180,E1 17714.782,E2 17714.782} C_VEL
LIN {X 0,Y 390.997,Z 1162.909,A -85,B 0,C 180,E1 17711.667,E2 17711.667} C_VEL
LIN {X 0,Y 394.535,Z 1153.069,A -85,B 0,C 180,E1 17708.284,E2 17708.284} C_VEL
LIN {X 0,Y 399.872,Z 1139.485,A -85,B 0,C 180,E1 17704.369,E2 17704.369} C_VEL
LIN {X 0,Y 404.672,Z 1127.923,A -85,B 0,C 180,E1 17701.52,E2 17701.52} C_VEL
LIN {X 0,Y 409.935,Z 1115.658,A -85,B 0,C 180,E1 17698.863,E2 17698.863} C_VEL
LIN {X 0,Y 415.882,Z 1101.998,A -85,B 0,C 180,E1 17696.264,E2 17696.264} C_VEL
LIN {X 0,Y 423.606,Z 1084.277,A -85,B 0,C 180,E1 17693.333,E2 17693.333} C_VEL
LIN {X 0,Y 431.162,Z 1066.313,A -85,B 0,C 180,E1 17690.808,E2 17690.808} C_VEL
LIN {X 0,Y 437.894,Z 1049.945,A -85,B 0,C 180,E1 17688.796,E2 17688.796} C_VEL
LIN {X 0,Y 444.388,Z 1033.556,A -85,B 0,C 180,E1 17687.02,E2 17687.02} C_VEL
LIN {X 0,Y 451.484,Z 1014.764,A -85,B 0,C 180,E1 17685.232,E2 17685.232} C_VEL
LIN {X 0,Y 459.98,Z 990.555,A -85,B 0,C 180,E1 17683.266,E2 17683.266} C_VEL
LIN {X 0,Y 466.496,Z 970.165,A -85,B 0,C 180,E1 17681.858,E2 17681.858} C_VEL
LIN {X 0,Y 472.16,Z 950.889,A -85,B 0,C 180,E1 17680.702,E2 17680.702} C_VEL
LIN {X 0,Y 477.449,Z 931.176,A -85,B 0,C 180,E1 17679.682,E2 17679.682} C_VEL
LIN {X 0,Y 482.711,Z 909.23,A -85,B 0,C 180,E1 17678.711,E2 17678.711} C_VEL
LIN {X 0,Y 488.485,Z 880.723,A -85,B 0,C 180,E1 17677.687,E2 17677.687} C_VEL
LIN {X 0,Y 492.233,Z 858.042,A -85,B 0,C 180,E1 17677.045,E2 17677.045} C_VEL
LIN {X 0,Y 495.121,Z 836.463,A -85,B 0,C 180,E1 17676.559,E2 17676.559} C_VEL
LIN {X 0,Y 497.365,Z 813.232,A -85,B 0,C 180,E1 17676.14,E2 17676.14} C_VEL
LIN {X 0,Y 511.116,Z 596.254,A -85,B 0,C 180,E1 17672.759,E2 17672.759} C_VEL
LIN {X 0,Y 516.277,Z 516.161,A -85,B 0,C 180,E1 17671.496,E2 17671.496} C_VEL
LIN {X 0,Y 506.18,Z 500.884,A -85,B 0,C 180,E1 17668.686,E2 17668.686} C_VEL
LIN {X 0,Y 497.793,Z 488.797,A -85,B 0,C 180,E1 17666.033,E2 17666.033} C_VEL
LIN {X 0,Y 491.303,Z 479.801,A -85,B 0,C 180,E1 17663.7,E2 17663.7} C_VEL
LIN {X 0,Y 487.618,Z 474.856,A -85,B 0,C 180,E1 17662.23,E2 17662.23} C_VEL
LIN {X 0,Y 484.209,Z 470.291,A -85,B 0,C 180,E1 17660.741,E2 17660.741} C_VEL
LIN {X 0,Y 480.513,Z 465.314,A -85,B 0,C 180,E1 17658.943,E2 17658.943} C_VEL
LIN {X 0,Y 476.716,Z 460.347,A -85,B 0,C 180,E1 17656.825,E2 17656.825} C_VEL
LIN {X 0,Y 473.552,Z 456.498,A -85,B 0,C 180,E1 17654.756,E2 17654.756} C_VEL
LIN {X 0,Y 472.53,Z 454.813,A -85,B 0,C 180,E1 17653.959,E2 17653.959} C_VEL
LIN {X 0,Y 469.612,Z 451.791,A -85,B 0,C 180,E1 17651.421,E2 17651.421} C_VEL
LIN {X 0,Y 468.267,Z 448.99,A -85,B 0,C 180,E1 17649.712,E2 17649.712} C_VEL
LIN {X 0,Y 465.828,Z 447.426,A -85,B 0,C 180,E1 17644.062,E2 17644.062} C_VEL
LIN {X 0,Y 466.597,Z 448.102,A -85,B 0,C 180,E1 17640,E2 17640} C_VEL
LIN {X 0,Y 468.514,Z 449.349,A -85,B 0,C 180,E1 17637.064,E2 17637.064} C_VEL
LIN {X 0,Y 470.538,Z 453.112,A -85,B 0,C 180,E1 17634.757,E2 17634.757} C_VEL
LIN {X 0,Y 473.008,Z 455.462,A -85,B 0,C 180,E1 17632.774,E2 17632.774} C_VEL
LIN {X 0,Y 476.022,Z 459.657,A -85,B 0,C 180,E1 17630.692,E2 17630.692} C_VEL
LIN {X 0,Y 477.519,Z 461.277,A -85,B 0,C 180,E1 17629.809,E2 17629.809} C_VEL
LIN {X 0,Y 481.868,Z 467.135,A -85,B 0,C 180,E1 17627.476,E2 17627.476} C_VEL
LIN {X 0,Y 486.351,Z 473.103,A -85,B 0,C 180,E1 17625.413,E2 17625.413} C_VEL
LIN {X 0,Y 490.335,Z 478.508,A -85,B 0,C 180,E1 17623.777,E2 17623.777} C_VEL
LIN {X 0,Y 496.683,Z 487.135,A -85,B 0,C 180,E1 17621.453,E2 17621.453} C_VEL
LIN {X 0,Y 503.555,Z 497.08,A -85,B 0,C 180,E1 17619.21,E2 17619.21} C_VEL
LIN {X 0,Y 513.811,Z 513.925,A -85,B 0,C 180,E1 17616.214,E2 17616.214} C_VEL
LIN {X 0,Y 516.303,Z 518.576,A -85,B 0,C 180,E1 17615.531,E2 17615.531} C_VEL
LIN {X 0,Y 502.38,Z 735.945,A -85,B 0,C 180,E1 17612.149,E2 17612.149} C_VEL
LIN {X 0,Y 496.603,Z 825.888,A -85,B 0,C 180,E1 17610.731,E2 17610.731} C_VEL
LIN {X 0,Y 493.493,Z 853.881,A -85,B 0,C 180,E1 17610.189,E2 17610.189} C_VEL
LIN {X 0,Y 489.426,Z 879.526,A -85,B 0,C 180,E1 17609.525,E2 17609.525} C_VEL
LIN {X 0,Y 485.451,Z 900.556,A -85,B 0,C 180,E1 17608.846,E2 17608.846} C_VEL
LIN {X 0,Y 481.006,Z 920.897,A -85,B 0,C 180,E1 17608.062,E2 17608.062} C_VEL
LIN {X 0,Y 475.778,Z 942.118,A -85,B 0,C 180,E1 17607.093,E2 17607.093} C_VEL
LIN {X 0,Y 468.555,Z 968.145,A -85,B 0,C 180,E1 17605.672,E2 17605.672} C_VEL
LIN {X 0,Y 461.635,Z 990.162,A -85,B 0,C 180,E1 17604.236,E2 17604.236} C_VEL
LIN {X 0,Y 455.394,Z 1008.621,A -85,B 0,C 180,E1 17602.844,E2 17602.844} C_VEL
LIN {X 0,Y 448.73,Z 1027.149,A -85,B 0,C 180,E1 17601.248,E2 17601.248} C_VEL
LIN {X 0,Y 440.741,Z 1048.223,A -85,B 0,C 180,E1 17599.163,E2 17599.163} C_VEL
LIN {X 0,Y 432.384,Z 1068.797,A -85,B 0,C 180,E1 17596.754,E2 17596.754} C_VEL
LIN {X 0,Y 425.726,Z 1084.756,A -85,B 0,C 180,E1 17594.606,E2 17594.606} C_VEL
LIN {X 0,Y 419.487,Z 1099.467,A -85,B 0,C 180,E1 17592.36,E2 17592.36} C_VEL
LIN {X 0,Y 412.76,Z 1115.271,A -85,B 0,C 180,E1 17589.615,E2 17589.615} C_VEL
LIN {X 0,Y 405.773,Z 1131.772,A -85,B 0,C 180,E1 17586.255,E2 17586.255} C_VEL
LIN {X 0,Y 400.597,Z 1144.245,A -85,B 0,C 180,E1 17583.305,E2 17583.305} C_VEL
LIN {X 0,Y 396.329,Z 1155.116,A -85,B 0,C 180,E1 17580.364,E2 17580.364} C_VEL
LIN {X 0,Y 392.376,Z 1166.008,A -85,B 0,C 180,E1 17576.974,E2 17576.974} C_VEL
LIN {X 0,Y 388.793,Z 1177.044,A -85,B 0,C 180,E1 17572.85,E2 17572.85} C_VEL
LIN {X 0,Y 386.817,Z 1184.206,A -85,B 0,C 180,E1 17569.635,E2 17569.635} C_VEL
LIN {X 0,Y 385.457,Z 1190.207,A -85,B 0,C 180,E1 17566.424,E2 17566.424} C_VEL
LIN {X 0,Y 384.634,Z 1194.884,A -85,B 0,C 180,E1 17563.377,E2 17563.377} C_VEL
LIN {X 0,Y 384.172,Z 1198.741,A -85,B 0,C 180,E1 17560.194,E2 17560.194} C_VEL
LIN {X 0,Y 383.971,Z 1201.547,A -85,B 0,C 180,E1 17557.03,E2 17557.03} C_VEL
LIN {X 0,Y 383.916,Z 1203.325,A -85,B 0,C 180,E1 17553.883,E2 17553.883} C_VEL
LIN {X 0,Y 383.903,Z 1204.134,A -85,B 0,C 180,E1 17550.448,E2 17550.448} C_VEL
LIN {X 0,Y 383.915,Z 1203.631,A -85,B 0,C 180,E1 17546.715,E2 17546.715} C_VEL
LIN {X 0,Y 383.967,Z 1201.721,A -85,B 0,C 180,E1 17543.12,E2 17543.12} C_VEL
LIN {X 0,Y 384.174,Z 1198.845,A -85,B 0,C 180,E1 17539.806,E2 17539.806} C_VEL
LIN {X 0,Y 384.638,Z 1195.059,A -85,B 0,C 180,E1 17536.623,E2 17536.623} C_VEL
LIN {X 0,Y 385.47,Z 1190.48,A -85,B 0,C 180,E1 17533.577,E2 17533.577} C_VEL
LIN {X 0,Y 386.843,Z 1184.62,A -85,B 0,C 180,E1 17530.366,E2 17530.366} C_VEL
LIN {X 0,Y 388.845,Z 1177.652,A -85,B 0,C 180,E1 17527.153,E2 17527.153} C_VEL
LIN {X 0,Y 392.173,Z 1167.916,A -85,B 0,C 180,E1 17523.339,E2 17523.339} C_VEL
LIN {X 0,Y 396.628,Z 1156.247,A -85,B 0,C 180,E1 17519.556,E2 17519.556} C_VEL
LIN {X 0,Y 401.338,Z 1145.012,A -85,B 0,C 180,E1 17516.422,E2 17516.422} C_VEL
LIN {X 0,Y 406.691,Z 1132.976,A -85,B 0,C 180,E1 17513.49,E2 17513.49} C_VEL
LIN {X 0,Y 413.86,Z 1117.429,A -85,B 0,C 180,E1 17510.192,E2 17510.192} C_VEL
LIN {X 0,Y 421.894,Z 1100.007,A -85,B 0,C 180,E1 17507.083,E2 17507.083} C_VEL
LIN {X 0,Y 428.77,Z 1085.131,A -85,B 0,C 180,E1 17504.77,E2 17504.77} C_VEL
LIN {X 0,Y 436.01,Z 1069.239,A -85,B 0,C 180,E1 17502.599,E2 17502.599} C_VEL
LIN {X 0,Y 445.037,Z 1048.966,A -85,B 0,C 180,E1 17500.193,E2 17500.193} C_VEL
LIN {X 0,Y 453.94,Z 1027.534,A -85,B 0,C 180,E1 17498.054,E2 17498.054} C_VEL
LIN {X 0,Y 461.206,Z 1009.074,A -85,B 0,C 180,E1 17496.458,E2 17496.458} C_VEL
LIN {X 0,Y 468.128,Z 990.369,A -85,B 0,C 180,E1 17495.046,E2 17495.046} C_VEL
LIN {X 0,Y 475.283,Z 969.599,A -85,B 0,C 180,E1 17493.694,E2 17493.694} C_VEL
LIN {X 0,Y 483.478,Z 942.94,A -85,B 0,C 180,E1 17492.239,E2 17492.239} C_VEL
LIN {X 0,Y 489.427,Z 920.903,A -85,B 0,C 180,E1 17491.245,E2 17491.245} C_VEL
LIN {X 0,Y 494.246,Z 900.761,A -85,B 0,C 180,E1 17490.481,E2 17490.481} C_VEL
LIN {X 0,Y 498.617,Z 879.633,A -85,B 0,C 180,E1 17489.81,E2 17489.81} C_VEL
LIN {X 0,Y 502.794,Z 855.601,A -85,B 0,C 180,E1 17489.199,E2 17489.199} C_VEL
LIN {X 0,Y 506.456,Z 826.507,A -85,B 0,C 180,E1 17488.635,E2 17488.635} C_VEL
LIN {X 0,Y 511.763,Z 755.096,A -85,B 0,C 180,E1 17487.501,E2 17487.501} C_VEL
LIN {X 0,Y 527.882,Z 536.413,A -85,B 0,C 180,E1 17484.092,E2 17484.092} C_VEL
LIN {X 0,Y 528.771,Z 523.684,A -85,B 0,C 180,E1 17483.87,E2 17483.87} C_VEL
LIN {X 0,Y 520.652,Z 510.092,A -85,B 0,C 180,E1 17480.811,E2 17480.811} C_VEL
LIN {X 0,Y 515.726,Z 502.823,A -85,B 0,C 180,E1 17478.657,E2 17478.657} C_VEL
LIN {X 0,Y 512.592,Z 498.371,A -85,B 0,C 180,E1 17477.101,E2 17477.101} C_VEL
LIN {X 0,Y 509.353,Z 493.668,A -85,B 0,C 180,E1 17475.251,E2 17475.251} C_VEL
LIN {X 0,Y 505.785,Z 488.732,A -85,B 0,C 180,E1 17472.792,E2 17472.792} C_VEL
LIN {X 0,Y 502.698,Z 484.393,A -85,B 0,C 180,E1 17469.907,E2 17469.907} C_VEL
LIN {X 0,Y 502.208,Z 483.4,A -85,B 0,C 180,E1 17469.281,E2 17469.281} C_VEL
LIN {X 0,Y 499.794,Z 481.274,A -85,B 0,C 180,E1 17464.015,E2 17464.015} C_VEL
LIN {X 0,Y 500.184,Z 481.809,A -85,B 0,C 180,E1 17460.916,E2 17460.916} C_VEL
LIN {X 0,Y 502.415,Z 483.659,A -85,B 0,C 180,E1 17457.262,E2 17457.262} C_VEL
LIN {X 0,Y 504.94,Z 487.919,A -85,B 0,C 180,E1 17454.66,E2 17454.66} C_VEL
LIN {X 0,Y 506.399,Z 489.517,A -85,B 0,C 180,E1 17453.538,E2 17453.538} C_VEL
LIN {X 0,Y 510.378,Z 495.152,A -85,B 0,C 180,E1 17450.926,E2 17450.926} C_VEL
LIN {X 0,Y 514.149,Z 500.554,A -85,B 0,C 180,E1 17448.899,E2 17448.899} C_VEL
LIN {X 0,Y 518.098,Z 506.259,A -85,B 0,C 180,E1 17447.063,E2 17447.063} C_VEL
LIN {X 0,Y 523.331,Z 513.857,A -85,B 0,C 180,E1 17444.939,E2 17444.939} C_VEL
LIN {X 0,Y 528.832,Z 522.305,A -85,B 0,C 180,E1 17442.958,E2 17442.958} C_VEL
LIN {X 0,Y 512.949,Z 736.483,A -85,B 0,C 180,E1 17439.62,E2 17439.62} C_VEL
LIN {X 0,Y 506.714,Z 820.834,A -85,B 0,C 180,E1 17438.286,E2 17438.286} C_VEL
LIN {X 0,Y 503.276,Z 848.983,A -85,B 0,C 180,E1 17437.742,E2 17437.742} C_VEL
LIN {X 0,Y 499.015,Z 873.913,A -85,B 0,C 180,E1 17437.099,E2 17437.099} C_VEL
LIN {X 0,Y 494.676,Z 895.044,A -85,B 0,C 180,E1 17436.424,E2 17436.424} C_VEL
LIN {X 0,Y 489.906,Z 915.168,A -85,B 0,C 180,E1 17435.652,E2 17435.652} C_VEL
LIN {X 0,Y 484.273,Z 936.191,A -85,B 0,C 180,E1 17434.697,E2 17434.697} C_VEL
LIN {X 0,Y 476.643,Z 961.457,A -85,B 0,C 180,E1 17433.332,E2 17433.332} C_VEL
LIN {X 0,Y 468.893,Z 983.996,A -85,B 0,C 180,E1 17431.865,E2 17431.865} C_VEL
LIN {X 0,Y 461.795,Z 1003.122,A -85,B 0,C 180,E1 17430.418,E2 17430.418} C_VEL
LIN {X 0,Y 454.291,Z 1022.084,A -85,B 0,C 180,E1 17428.766,E2 17428.766} C_VEL
LIN {X 0,Y 445.136,Z 1043.863,A -85,B 0,C 180,E1 17426.559,E2 17426.559} C_VEL
LIN {X 0,Y 436.548,Z 1063.016,A -85,B 0,C 180,E1 17424.263,E2 17424.263} C_VEL
LIN {X 0,Y 429.391,Z 1078.538,A -85,B 0,C 180,E1 17422.127,E2 17422.127} C_VEL
LIN {X 0,Y 422.551,Z 1093.132,A -85,B 0,C 180,E1 17419.844,E2 17419.844} C_VEL
LIN {X 0,Y 414.864,Z 1109.525,A -85,B 0,C 180,E1 17416.908,E2 17416.908} C_VEL
LIN {X 0,Y 407.5,Z 1125.192,A -85,B 0,C 180,E1 17413.588,E2 17413.588} C_VEL
LIN {X 0,Y 402.041,Z 1137.152,A -85,B 0,C 180,E1 17410.661,E2 17410.661} C_VEL
LIN {X 0,Y 397.428,Z 1147.78,A -85,B 0,C 180,E1 17407.687,E2 17407.687} C_VEL
LIN {X 0,Y 393.109,Z 1158.581,A -85,B 0,C 180,E1 17404.201,E2 17404.201} C_VEL
LIN {X 0,Y 389.254,Z 1169.298,A -85,B 0,C 180,E1 17400.041,E2 17400.041} C_VEL
LIN {X 0,Y 387.072,Z 1176.446,A -85,B 0,C 180,E1 17396.709,E2 17396.709} C_VEL
LIN {X 0,Y 385.646,Z 1182.169,A -85,B 0,C 180,E1 17393.533,E2 17393.533} C_VEL
LIN {X 0,Y 384.727,Z 1186.834,A -85,B 0,C 180,E1 17390.38,E2 17390.38} C_VEL
LIN {X 0,Y 384.238,Z 1190.493,A -85,B 0,C 180,E1 17387.246,E2 17387.246} C_VEL
LIN {X 0,Y 384.004,Z 1193.148,A -85,B 0,C 180,E1 17384.167,E2 17384.167} C_VEL
LIN {X 0,Y 383.925,Z 1194.861,A -85,B 0,C 180,E1 17381.111,E2 17381.111} C_VEL
LIN {X 0,Y 383.909,Z 1195.644,A -85,B 0,C 180,E1 17378.085,E2 17378.085} C_VEL
LIN {X 0,Y 383.916,Z 1195.494,A -85,B 0,C 180,E1 17374.93,E2 17374.93} C_VEL
LIN {X 0,Y 383.947,Z 1194.155,A -85,B 0,C 180,E1 17371.343,E2 17371.343} C_VEL
LIN {X 0,Y 384.15,Z 1191.181,A -85,B 0,C 180,E1 17367.464,E2 17367.464} C_VEL
LIN {X 0,Y 384.615,Z 1187.274,A -85,B 0,C 180,E1 17364.031,E2 17364.031} C_VEL
LIN {X 0,Y 385.324,Z 1183.25,A -85,B 0,C 180,E1 17361.242,E2 17361.242} C_VEL
LIN {X 0,Y 384.725,Z 1181.481,A -85,B 0,C 180,E1 17360.123,E2 17360.123} C_VEL
LIN {X 0,Y 379.777,Z 1176.382,A -85,B 0,C 180,E1 17357.027,E2 17357.027} C_VEL
LIN {X 0,Y 379.653,Z 1174.696,A -85,B 0,C 180,E1 17356.136,E2 17356.136} C_VEL
LIN {X 0,Y 382.671,Z 1165.173,A -85,B 0,C 180,E1 17352.01,E2 17352.01} C_VEL
LIN {X 0,Y 385.973,Z 1156.154,A -85,B 0,C 180,E1 17348.736,E2 17348.736} C_VEL
LIN {X 0,Y 389.73,Z 1146.712,A -85,B 0,C 180,E1 17345.765,E2 17345.765} C_VEL
LIN {X 0,Y 394.503,Z 1135.51,A -85,B 0,C 180,E1 17342.694,E2 17342.694} C_VEL
LIN {X 0,Y 401.227,Z 1120.289,A -85,B 0,C 180,E1 17339.113,E2 17339.113} C_VEL
LIN {X 0,Y 407.816,Z 1105.584,A -85,B 0,C 180,E1 17336.183,E2 17336.183} C_VEL
LIN {X 0,Y 414.127,Z 1091.545,A -85,B 0,C 180,E1 17333.735,E2 17333.735} C_VEL
LIN {X 0,Y 420.868,Z 1076.381,A -85,B 0,C 180,E1 17331.411,E2 17331.411} C_VEL
LIN {X 0,Y 429.467,Z 1056.654,A -85,B 0,C 180,E1 17328.787,E2 17328.787} C_VEL
LIN {X 0,Y 437.619,Z 1036.758,A -85,B 0,C 180,E1 17326.551,E2 17326.551} C_VEL
LIN {X 0,Y 444.348,Z 1019.565,A -85,B 0,C 180,E1 17324.863,E2 17324.863} C_VEL
LIN {X 0,Y 450.893,Z 1001.881,A -85,B 0,C 180,E1 17323.336,E2 17323.336} C_VEL
LIN {X 0,Y 457.73,Z 982.168,A -85,B 0,C 180,E1 17321.852,E2 17321.852} C_VEL
LIN {X 0,Y 465.668,Z 957.049,A -85,B 0,C 180,E1 17320.243,E2 17320.243} C_VEL
LIN {X 0,Y 471.884,Z 934.798,A -85,B 0,C 180,E1 17319.053,E2 17319.053} C_VEL
LIN {X 0,Y 476.819,Z 915.12,A -85,B 0,C 180,E1 17318.155,E2 17318.155} C_VEL
LIN {X 0,Y 481.407,Z 894.401,A -85,B 0,C 180,E1 17317.35,E2 17317.35} C_VEL
LIN {X 0,Y 485.598,Z 872.467,A -85,B 0,C 180,E1 17316.641,E2 17316.641} C_VEL
LIN {X 0,Y 489.899,Z 844.777,A -85,B 0,C 180,E1 17315.935,E2 17315.935} C_VEL
LIN {X 0,Y 492.69,Z 819.181,A -85,B 0,C 180,E1 17315.449,E2 17315.449} C_VEL
LIN {X 0,Y 504.289,Z 642.253,A -85,B 0,C 180,E1 17312.678,E2 17312.678} C_VEL
LIN {X 0,Y 512.357,Z 520.936,A -85,B 0,C 180,E1 17310.781,E2 17310.781} C_VEL
LIN {X 0,Y 502.98,Z 506.627,A -85,B 0,C 180,E1 17308.076,E2 17308.076} C_VEL
LIN {X 0,Y 494.126,Z 493.602,A -85,B 0,C 180,E1 17305.147,E2 17305.147} C_VEL
LIN {X 0,Y 486.799,Z 483.425,A -85,B 0,C 180,E1 17302.333,E2 17302.333} C_VEL
LIN {X 0,Y 482.364,Z 477.556,A -85,B 0,C 180,E1 17300.38,E2 17300.38} C_VEL
LIN {X 0,Y 478.981,Z 472.896,A -85,B 0,C 180,E1 17298.689,E2 17298.689} C_VEL
LIN {X 0,Y 475.357,Z 468.072,A -85,B 0,C 180,E1 17296.623,E2 17296.623} C_VEL
LIN {X 0,Y 472.157,Z 464.027,A -85,B 0,C 180,E1 17294.471,E2 17294.471} C_VEL
LIN {X 0,Y 471.247,Z 462.594,A -85,B 0,C 180,E1 17293.747,E2 17293.747} C_VEL
LIN {X 0,Y 468.414,Z 459.505,A -85,B 0,C 180,E1 17291.201,E2 17291.201} C_VEL
LIN {X 0,Y 467.201,Z 456.9,A -85,B 0,C 180,E1 17289.61,E2 17289.61} C_VEL
LIN {X 0,Y 464.845,Z 455.363,A -85,B 0,C 180,E1 17283.947,E2 17283.947} C_VEL
LIN {X 0,Y 465.796,Z 456.164,A -85,B 0,C 180,E1 17279.631,E2 17279.631} C_VEL
LIN {X 0,Y 467.43,Z 457.261,A -85,B 0,C 180,E1 17277.18,E2 17277.18} C_VEL
LIN {X 0,Y 469.554,Z 461.131,A -85,B 0,C 180,E1 17274.746,E2 17274.746} C_VEL
LIN {X 0,Y 471.706,Z 463.139,A -85,B 0,C 180,E1 17272.999,E2 17272.999} C_VEL
LIN {X 0,Y 474.651,Z 467.352,A -85,B 0,C 180,E1 17270.91,E2 17270.91} C_VEL
LIN {X 0,Y 476.123,Z 468.971,A -85,B 0,C 180,E1 17270.023,E2 17270.023} C_VEL
LIN {X 0,Y 480.399,Z 474.842,A -85,B 0,C 180,E1 17267.682,E2 17267.682} C_VEL
LIN {X 0,Y 484.694,Z 480.634,A -85,B 0,C 180,E1 17265.667,E2 17265.667} C_VEL
LIN {X 0,Y 488.758,Z 486.246,A -85,B 0,C 180,E1 17263.968,E2 17263.968} C_VEL
LIN {X 0,Y 494.955,Z 494.845,A -85,B 0,C 180,E1 17261.661,E2 17261.661} C_VEL
LIN {X 0,Y 501.328,Z 504.208,A -85,B 0,C 180,E1 17259.541,E2 17259.541} C_VEL
LIN {X 0,Y 511.34,Z 520.949,A -85,B 0,C 180,E1 17256.551,E2 17256.551} C_VEL
LIN {X 0,Y 512.355,Z 523.067,A -85,B 0,C 180,E1 17256.258,E2 17256.258} C_VEL
LIN {X 0,Y 498.064,Z 740.12,A -85,B 0,C 180,E1 17252.878,E2 17252.878} C_VEL
LIN {X 0,Y 492.396,Z 825.799,A -85,B 0,C 180,E1 17251.524,E2 17251.524} C_VEL
LIN {X 0,Y 489.223,Z 853.78,A -85,B 0,C 180,E1 17250.983,E2 17250.983} C_VEL
LIN {X 0,Y 485.054,Z 879.49,A -85,B 0,C 180,E1 17250.321,E2 17250.321} C_VEL
LIN {X 0,Y 480.924,Z 900.836,A -85,B 0,C 180,E1 17249.632,E2 17249.632} C_VEL
LIN {X 0,Y 476.224,Z 921.794,A -85,B 0,C 180,E1 17248.822,E2 17248.822} C_VEL
LIN {X 0,Y 470.132,Z 945.798,A -85,B 0,C 180,E1 17247.713,E2 17247.713} C_VEL
LIN {X 0,Y 462.748,Z 971.057,A -85,B 0,C 180,E1 17246.291,E2 17246.291} C_VEL
LIN {X 0,Y 456.449,Z 990.515,A -85,B 0,C 180,E1 17245.01,E2 17245.01} C_VEL
LIN {X 0,Y 449.851,Z 1009.488,A -85,B 0,C 180,E1 17243.571,E2 17243.571} C_VEL
LIN {X 0,Y 442.783,Z 1028.55,A -85,B 0,C 180,E1 17241.912,E2 17241.912} C_VEL
LIN {X 0,Y 433.587,Z 1051.755,A -85,B 0,C 180,E1 17239.551,E2 17239.551} C_VEL
LIN {X 0,Y 426.201,Z 1069.386,A -85,B 0,C 180,E1 17237.445,E2 17237.445} C_VEL
LIN {X 0,Y 419.339,Z 1085.285,A -85,B 0,C 180,E1 17235.279,E2 17235.279} C_VEL
LIN {X 0,Y 412.637,Z 1100.546,A -85,B 0,C 180,E1 17232.913,E2 17232.913} C_VEL
LIN {X 0,Y 404.87,Z 1118.157,A -85,B 0,C 180,E1 17229.763,E2 17229.763} C_VEL
LIN {X 0,Y 398.405,Z 1132.775,A -85,B 0,C 180,E1 17226.676,E2 17226.676} C_VEL
LIN {X 0,Y 393.325,Z 1144.561,A -85,B 0,C 180,E1 17223.829,E2 17223.829} C_VEL
LIN {X 0,Y 389.002,Z 1155.068,A -85,B 0,C 180,E1 17220.935,E2 17220.935} C_VEL
LIN {X 0,Y 384.923,Z 1165.788,A -85,B 0,C 180,E1 17217.54,E2 17217.54} C_VEL
LIN {X 0,Y 381.111,Z 1176.888,A -85,B 0,C 180,E1 17213.325,E2 17213.325} C_VEL
LIN {X 0,Y 379.034,Z 1184.042,A -85,B 0,C 180,E1 17210.055,E2 17210.055} C_VEL
LIN {X 0,Y 377.567,Z 1190.059,A -85,B 0,C 180,E1 17206.777,E2 17206.777} C_VEL
LIN {X 0,Y 376.697,Z 1194.751,A -85,B 0,C 180,E1 17203.664,E2 17203.664} C_VEL
LIN {X 0,Y 376.209,Z 1198.458,A -85,B 0,C 180,E1 17200.567,E2 17200.567} C_VEL
LIN {X 0,Y 375.999,Z 1201.207,A -85,B 0,C 180,E1 17197.487,E2 17197.487} C_VEL
LIN {X 0,Y 375.919,Z 1203.019,A -85,B 0,C 180,E1 17194.424,E2 17194.424} C_VEL
LIN {X 0,Y 375.914,Z 1203.884,A -85,B 0,C 180,E1 17191.524,E2 17191.524} C_VEL
LIN {X 0,Y 375.915,Z 1203.924,A -85,B 0,C 180,E1 17188.628,E2 17188.628} C_VEL
LIN {X 0,Y 375.918,Z 1203.073,A -85,B 0,C 180,E1 17185.576,E2 17185.576} C_VEL
LIN {X 0,Y 375.999,Z 1201.31,A -85,B 0,C 180,E1 17182.513,E2 17182.513} C_VEL
LIN {X 0,Y 376.211,Z 1198.627,A -85,B 0,C 180,E1 17179.433,E2 17179.433} C_VEL
LIN {X 0,Y 376.741,Z 1194.806,A -85,B 0,C 180,E1 17176.181,E2 17176.181} C_VEL
LIN {X 0,Y 377.639,Z 1190.194,A -85,B 0,C 180,E1 17173.068,E2 17173.068} C_VEL
LIN {X 0,Y 379.156,Z 1184.301,A -85,B 0,C 180,E1 17169.79,E2 17169.79} C_VEL
LIN {X 0,Y 381.427,Z 1176.949,A -85,B 0,C 180,E1 17166.355,E2 17166.355} C_VEL
LIN {X 0,Y 385.398,Z 1166.186,A -85,B 0,C 180,E1 17162.161,E2 17162.161} C_VEL
LIN {X 0,Y 389.852,Z 1155.285,A -85,B 0,C 180,E1 17158.625,E2 17158.625} C_VEL
LIN {X 0,Y 394.652,Z 1144.531,A -85,B 0,C 180,E1 17155.6,E2 17155.6} C_VEL
LIN {X 0,Y 399.976,Z 1133.088,A -85,B 0,C 180,E1 17152.775,E2 17152.775} C_VEL
LIN {X 0,Y 407.112,Z 1118.27,A -85,B 0,C 180,E1 17149.581,E2 17149.581} C_VEL
LIN {X 0,Y 415.7,Z 1100.481,A -85,B 0,C 180,E1 17146.346,E2 17146.346} C_VEL
LIN {X 0,Y 422.772,Z 1085.774,A -85,B 0,C 180,E1 17144.031,E2 17144.031} C_VEL
LIN {X 0,Y 429.985,Z 1070.51,A -85,B 0,C 180,E1 17141.918,E2 17141.918} C_VEL
LIN {X 0,Y 437.726,Z 1053.661,A -85,B 0,C 180,E1 17139.871,E2 17139.871} C_VEL
LIN {X 0,Y 447.243,Z 1032.101,A -85,B 0,C 180,E1 17137.614,E2 17137.614} C_VEL
LIN {X 0,Y 455.855,Z 1010.983,A -85,B 0,C 180,E1 17135.753,E2 17135.753} C_VEL
LIN {X 0,Y 463.177,Z 991.836,A -85,B 0,C 180,E1 17134.294,E2 17134.294} C_VEL
LIN {X 0,Y 469.949,Z 972.839,A -85,B 0,C 180,E1 17133.042,E2 17133.042} C_VEL
LIN {X 0,Y 476.733,Z 952.01,A -85,B 0,C 180,E1 17131.853,E2 17131.853} C_VEL
LIN {X 0,Y 484.382,Z 925.573,A -85,B 0,C 180,E1 17130.597,E2 17130.597} C_VEL
LIN {X 0,Y 489.963,Z 903.152,A -85,B 0,C 180,E1 17129.729,E2 17129.729} C_VEL
LIN {X 0,Y 494.563,Z 881.734,A -85,B 0,C 180,E1 17129.041,E2 17129.041} C_VEL
LIN {X 0,Y 498.452,Z 860.311,A -85,B 0,C 180,E1 17128.482,E2 17128.482} C_VEL
LIN {X 0,Y 501.98,Z 835.955,A -85,B 0,C 180,E1 17127.978,E2 17127.978} C_VEL
LIN {X 0,Y 505.209,Z 799.651,A -85,B 0,C 180,E1 17127.374,E2 17127.374} C_VEL
LIN {X 0,Y 521.72,Z 578.831,A -85,B 0,C 180,E1 17123.933,E2 17123.933} C_VEL
LIN {X 0,Y 525.545,Z 528.935,A -85,B 0,C 180,E1 17123.14,E2 17123.14} C_VEL
LIN {X 0,Y 518.76,Z 517.277,A -85,B 0,C 180,E1 17120.477,E2 17120.477} C_VEL
LIN {X 0,Y 514.059,Z 510.228,A -85,B 0,C 180,E1 17118.367,E2 17118.367} C_VEL
LIN {X 0,Y 511.046,Z 505.88,A -85,B 0,C 180,E1 17116.832,E2 17116.832} C_VEL
LIN {X 0,Y 507.834,Z 501.188,A -85,B 0,C 180,E1 17114.947,E2 17114.947} C_VEL
LIN {X 0,Y 504.522,Z 496.484,A -85,B 0,C 180,E1 17112.592,E2 17112.592} C_VEL
LIN {X 0,Y 501.491,Z 491.987,A -85,B 0,C 180,E1 17109.642,E2 17109.642} C_VEL
LIN {X 0,Y 501.046,Z 491.255,A -85,B 0,C 180,E1 17109.071,E2 17109.071} C_VEL
LIN {X 0,Y 498.818,Z 489.217,A -85,B 0,C 180,E1 17104.023,E2 17104.023} C_VEL
LIN {X 0,Y 499.167,Z 489.706,A -85,B 0,C 180,E1 17101.033,E2 17101.033} C_VEL
LIN {X 0,Y 501.333,Z 491.567,A -85,B 0,C 180,E1 17097.371,E2 17097.371} C_VEL
LIN {X 0,Y 503.955,Z 495.937,A -85,B 0,C 180,E1 17094.649,E2 17094.649} C_VEL
LIN {X 0,Y 505.25,Z 497.467,A -85,B 0,C 180,E1 17093.637,E2 17093.637} C_VEL
LIN {X 0,Y 509.004,Z 502.832,A -85,B 0,C 180,E1 17091.129,E2 17091.129} C_VEL
LIN {X 0,Y 512.707,Z 508.248,A -85,B 0,C 180,E1 17089.096,E2 17089.096} C_VEL
LIN {X 0,Y 516.598,Z 513.963,A -85,B 0,C 180,E1 17087.253,E2 17087.253} C_VEL
LIN {X 0,Y 521.689,Z 521.528,A -85,B 0,C 180,E1 17085.146,E2 17085.146} C_VEL
LIN {X 0,Y 525.585,Z 527.661,A -85,B 0,C 180,E1 17083.693,E2 17083.693} C_VEL
LIN {X 0,Y 509.203,Z 742.974,A -85,B 0,C 180,E1 17080.342,E2 17080.342} C_VEL
LIN {X 0,Y 503.246,Z 821.156,A -85,B 0,C 180,E1 17079.105,E2 17079.105} C_VEL
LIN {X 0,Y 499.677,Z 849.531,A -85,B 0,C 180,E1 17078.556,E2 17078.556} C_VEL
LIN {X 0,Y 495.379,Z 874.094,A -85,B 0,C 180,E1 17077.927,E2 17077.927} C_VEL
LIN {X 0,Y 491.063,Z 894.705,A -85,B 0,C 180,E1 17077.273,E2 17077.273} C_VEL
LIN {X 0,Y 486.217,Z 914.737,A -85,B 0,C 180,E1 17076.513,E2 17076.513} C_VEL
LIN {X 0,Y 480.612,Z 935.241,A -85,B 0,C 180,E1 17075.593,E2 17075.593} C_VEL
LIN {X 0,Y 473.206,Z 959.411,A -85,B 0,C 180,E1 17074.312,E2 17074.312} C_VEL
LIN {X 0,Y 464.885,Z 983.14,A -85,B 0,C 180,E1 17072.79,E2 17072.79} C_VEL
LIN {X 0,Y 457.521,Z 1002.513,A -85,B 0,C 180,E1 17071.334,E2 17071.334} C_VEL
LIN {X 0,Y 450.166,Z 1020.613,A -85,B 0,C 180,E1 17069.769,E2 17069.769} C_VEL
LIN {X 0,Y 442.312,Z 1038.863,A -85,B 0,C 180,E1 17067.962,E2 17067.962} C_VEL
LIN {X 0,Y 432.329,Z 1060.749,A -85,B 0,C 180,E1 17065.419,E2 17065.419} C_VEL
LIN {X 0,Y 424.266,Z 1077.618,A -85,B 0,C 180,E1 17063.117,E2 17063.117} C_VEL
LIN {X 0,Y 416.944,Z 1092.642,A -85,B 0,C 180,E1 17060.766,E2 17060.766} C_VEL
LIN {X 0,Y 409.274,Z 1108.283,A -85,B 0,C 180,E1 17057.959,E2 17057.959} C_VEL
LIN {X 0,Y 401.161,Z 1124.829,A -85,B 0,C 180,E1 17054.456,E2 17054.456} C_VEL
LIN {X 0,Y 395.413,Z 1136.832,A -85,B 0,C 180,E1 17051.491,E2 17051.491} C_VEL
LIN {X 0,Y 390.513,Z 1147.493,A -85,B 0,C 180,E1 17048.475,E2 17048.475} C_VEL
LIN {X 0,Y 386.279,Z 1157.388,A -85,B 0,C 180,E1 17045.255,E2 17045.255} C_VEL
LIN {X 0,Y 382.057,Z 1168.363,A -85,B 0,C 180,E1 17041.035,E2 17041.035} C_VEL
LIN {X 0,Y 379.414,Z 1176.307,A -85,B 0,C 180,E1 17037.293,E2 17037.293} C_VEL
LIN {X 0,Y 377.846,Z 1182.064,A -85,B 0,C 180,E1 17034.049,E2 17034.049} C_VEL
LIN {X 0,Y 376.844,Z 1186.764,A -85,B 0,C 180,E1 17030.826,E2 17030.826} C_VEL
LIN {X 0,Y 376.281,Z 1190.447,A -85,B 0,C 180,E1 17027.633,E2 17027.633} C_VEL
LIN {X 0,Y 376.026,Z 1193.147,A -85,B 0,C 180,E1 17024.474,E2 17024.474} C_VEL
LIN {X 0,Y 375.929,Z 1194.896,A -85,B 0,C 180,E1 17021.351,E2 17021.351} C_VEL
LIN {X 0,Y 375.915,Z 1195.706,A -85,B 0,C 180,E1 17018.317,E2 17018.317} C_VEL
LIN {X 0,Y 375.917,Z 1195.644,A -85,B 0,C 180,E1 17015.342,E2 17015.342} C_VEL
LIN {X 0,Y 375.931,Z 1194.699,A -85,B 0,C 180,E1 17012.286,E2 17012.286} C_VEL
LIN {X 0,Y 376.028,Z 1192.863,A -85,B 0,C 180,E1 17009.238,E2 17009.238} C_VEL
LIN {X 0,Y 376.279,Z 1190.135,A -85,B 0,C 180,E1 17006.191,E2 17006.191} C_VEL
LIN {X 0,Y 376.849,Z 1186.304,A -85,B 0,C 180,E1 17002.99,E2 17002.99} C_VEL
LIN {X 0,Y 377.962,Z 1180.964,A -85,B 0,C 180,E1 16999.483,E2 16999.483} C_VEL
LIN {X 0,Y 379.653,Z 1174.696,A -85,B 0,C 180,E1 16996.136,E2 16996.136} C_VEL
LIN {X 0,Y 379.375,Z 1172.523,A -85,B 0,C 180,E1 16995.012,E2 16995.012} C_VEL
LIN {X 0,Y 375.424,Z 1166.334,A -85,B 0,C 180,E1 16991.981,E2 16991.981} C_VEL
LIN {X 0,Y 375.545,Z 1164,A -85,B 0,C 180,E1 16991.026,E2 16991.026} C_VEL
LIN {X 0,Y 378.961,Z 1155.219,A -85,B 0,C 180,E1 16987.834,E2 16987.834} C_VEL
LIN {X 0,Y 383.479,Z 1144.649,A -85,B 0,C 180,E1 16984.519,E2 16984.519} C_VEL
LIN {X 0,Y 390.223,Z 1129.566,A -85,B 0,C 180,E1 16980.531,E2 16980.531} C_VEL
LIN {X 0,Y 396.164,Z 1116.758,A -85,B 0,C 180,E1 16977.652,E2 16977.652} C_VEL
LIN {X 0,Y 402.172,Z 1103.925,A -85,B 0,C 180,E1 16975.123,E2 16975.123} C_VEL
LIN {X 0,Y 408.869,Z 1089.569,A -85,B 0,C 180,E1 16972.636,E2 16972.636} C_VEL
LIN {X 0,Y 417.531,Z 1070.749,A -85,B 0,C 180,E1 16969.812,E2 16969.812} C_VEL
LIN {X 0,Y 425.941,Z 1051.504,A -85,B 0,C 180,E1 16967.373,E2 16967.373} C_VEL
LIN {X 0,Y 433.027,Z 1034.708,A -85,B 0,C 180,E1 16965.521,E2 16965.521} C_VEL
LIN {X 0,Y 439.778,Z 1017.866,A -85,B 0,C 180,E1 16963.887,E2 16963.887} C_VEL
LIN {X 0,Y 447.346,Z 997.85,A -85,B 0,C 180,E1 16962.189,E2 16962.189} C_VEL
LIN {X 0,Y 455.802,Z 973.363,A -85,B 0,C 180,E1 16960.431,E2 16960.431} C_VEL
LIN {X 0,Y 462.273,Z 952.56,A -85,B 0,C 180,E1 16959.168,E2 16959.168} C_VEL
LIN {X 0,Y 467.841,Z 932.905,A -85,B 0,C 180,E1 16958.143,E2 16958.143} C_VEL
LIN {X 0,Y 473.208,Z 911.704,A -85,B 0,C 180,E1 16957.196,E2 16957.196} C_VEL
LIN {X 0,Y 478.976,Z 885.503,A -85,B 0,C 180,E1 16956.225,E2 16956.225} C_VEL
LIN {X 0,Y 483.545,Z 859.354,A -85,B 0,C 180,E1 16955.475,E2 16955.475} C_VEL
LIN {X 0,Y 486.652,Z 837.291,A -85,B 0,C 180,E1 16954.977,E2 16954.977} C_VEL
LIN {X 0,Y 488.966,Z 814.698,A -85,B 0,C 180,E1 16954.567,E2 16954.567} C_VEL
LIN {X 0,Y 503.387,Z 599.935,A -85,B 0,C 180,E1 16951.21,E2 16951.21} C_VEL
LIN {X 0,Y 508.445,Z 525.715,A -85,B 0,C 180,E1 16950.039,E2 16950.039} C_VEL
LIN {X 0,Y 500.348,Z 513.176,A -85,B 0,C 180,E1 16947.622,E2 16947.622} C_VEL
LIN {X 0,Y 492.224,Z 500.986,A -85,B 0,C 180,E1 16944.866,E2 16944.866} C_VEL
LIN {X 0,Y 485.012,Z 490.823,A -85,B 0,C 180,E1 16942.037,E2 16942.037} C_VEL
LIN {X 0,Y 480.784,Z 485.118,A -85,B 0,C 180,E1 16940.133,E2 16940.133} C_VEL
LIN {X 0,Y 477.458,Z 480.477,A -85,B 0,C 180,E1 16938.435,E2 16938.435} C_VEL
LIN {X 0,Y 474.002,Z 475.794,A -85,B 0,C 180,E1 16936.42,E2 16936.42} C_VEL
LIN {X 0,Y 470.793,Z 471.592,A -85,B 0,C 180,E1 16934.2,E2 16934.2} C_VEL
LIN {X 0,Y 469.943,Z 470.353,A -85,B 0,C 180,E1 16933.513,E2 16933.513} C_VEL
LIN {X 0,Y 467.121,Z 467.022,A -85,B 0,C 180,E1 16930.858,E2 16930.858} C_VEL
LIN {X 0,Y 466.136,Z 464.81,A -85,B 0,C 180,E1 16929.507,E2 16929.507} C_VEL
LIN {X 0,Y 463.869,Z 463.304,A -85,B 0,C 180,E1 16923.955,E2 16923.955} C_VEL
LIN {X 0,Y 464.818,Z 464.108,A -85,B 0,C 180,E1 16919.63,E2 16919.63} C_VEL
LIN {X 0,Y 466.348,Z 465.172,A -85,B 0,C 180,E1 16917.296,E2 16917.296} C_VEL
LIN {X 0,Y 468.438,Z 469.002,A -85,B 0,C 180,E1 16914.857,E2 16914.857} C_VEL
LIN {X 0,Y 470.481,Z 470.964,A -85,B 0,C 180,E1 16913.165,E2 16913.165} C_VEL
LIN {X 0,Y 473.478,Z 475.233,A -85,B 0,C 180,E1 16911.009,E2 16911.009} C_VEL
LIN {X 0,Y 474.827,Z 476.826,A -85,B 0,C 180,E1 16910.179,E2 16910.179} C_VEL
LIN {X 0,Y 478.937,Z 482.545,A -85,B 0,C 180,E1 16907.888,E2 16907.888} C_VEL
LIN {X 0,Y 483.173,Z 488.35,A -85,B 0,C 180,E1 16905.866,E2 16905.866} C_VEL
LIN {X 0,Y 488.906,Z 496.245,A -85,B 0,C 180,E1 16903.484,E2 16903.484} C_VEL
LIN {X 0,Y 496.569,Z 507.413,A -85,B 0,C 180,E1 16900.717,E2 16900.717} C_VEL
LIN {X 0,Y 501.791,Z 515.929,A -85,B 0,C 180,E1 16899.012,E2 16899.012} C_VEL
LIN {X 0,Y 508.495,Z 527.454,A -85,B 0,C 180,E1 16896.998,E2 16896.998} C_VEL
LIN {X 0,Y 493.787,Z 744.906,A -85,B 0,C 180,E1 16893.609,E2 16893.609} C_VEL
LIN {X 0,Y 488.252,Z 826.046,A -85,B 0,C 180,E1 16892.324,E2 16892.324} C_VEL
LIN {X 0,Y 484.943,Z 854.328,A -85,B 0,C 180,E1 16891.775,E2 16891.775} C_VEL
LIN {X 0,Y 480.758,Z 879.564,A -85,B 0,C 180,E1 16891.127,E2 16891.127} C_VEL
LIN {X 0,Y 476.701,Z 900.124,A -85,B 0,C 180,E1 16890.467,E2 16890.467} C_VEL
LIN {X 0,Y 472,Z 920.705,A -85,B 0,C 180,E1 16889.68,E2 16889.68} C_VEL
LIN {X 0,Y 466.367,Z 942.515,A -85,B 0,C 180,E1 16888.688,E2 16888.688} C_VEL
LIN {X 0,Y 458.478,Z 969.356,A -85,B 0,C 180,E1 16887.214,E2 16887.214} C_VEL
LIN {X 0,Y 451.715,Z 989.809,A -85,B 0,C 180,E1 16885.877,E2 16885.877} C_VEL
LIN {X 0,Y 444.938,Z 1008.84,A -85,B 0,C 180,E1 16884.437,E2 16884.437} C_VEL
LIN {X 0,Y 437.904,Z 1027.343,A -85,B 0,C 180,E1 16882.831,E2 16882.831} C_VEL
LIN {X 0,Y 429.187,Z 1048.988,A -85,B 0,C 180,E1 16880.664,E2 16880.664} C_VEL
LIN {X 0,Y 420.366,Z 1069.323,A -85,B 0,C 180,E1 16878.24,E2 16878.24} C_VEL
LIN {X 0,Y 413.442,Z 1084.865,A -85,B 0,C 180,E1 16876.11,E2 16876.11} C_VEL
LIN {X 0,Y 406.485,Z 1100.157,A -85,B 0,C 180,E1 16873.725,E2 16873.725} C_VEL
LIN {X 0,Y 398.394,Z 1117.828,A -85,B 0,C 180,E1 16870.543,E2 16870.543} C_VEL
LIN {X 0,Y 391.648,Z 1132.473,A -85,B 0,C 180,E1 16867.416,E2 16867.416} C_VEL
LIN {X 0,Y 386.35,Z 1144.287,A -85,B 0,C 180,E1 16864.525,E2 16864.525} C_VEL
LIN {X 0,Y 381.8,Z 1154.817,A -85,B 0,C 180,E1 16861.585,E2 16861.585} C_VEL
LIN {X 0,Y 377.678,Z 1165.093,A -85,B 0,C 180,E1 16858.286,E2 16858.286} C_VEL
LIN {X 0,Y 373.607,Z 1176.312,A -85,B 0,C 180,E1 16854.003,E2 16854.003} C_VEL
LIN {X 0,Y 371.196,Z 1184.093,A -85,B 0,C 180,E1 16850.379,E2 16850.379} C_VEL
LIN {X 0,Y 369.691,Z 1189.906,A -85,B 0,C 180,E1 16847.145,E2 16847.145} C_VEL
LIN {X 0,Y 368.748,Z 1194.709,A -85,B 0,C 180,E1 16843.892,E2 16843.892} C_VEL
LIN {X 0,Y 368.216,Z 1198.496,A -85,B 0,C 180,E1 16840.641,E2 16840.641} C_VEL
LIN {X 0,Y 367.999,Z 1201.21,A -85,B 0,C 180,E1 16837.494,E2 16837.494} C_VEL
LIN {X 0,Y 367.919,Z 1202.986,A -85,B 0,C 180,E1 16834.364,E2 16834.364} C_VEL
LIN {X 0,Y 367.916,Z 1203.814,A -85,B 0,C 180,E1 16831.401,E2 16831.401} C_VEL
LIN {X 0,Y 367.914,Z 1203.818,A -85,B 0,C 180,E1 16828.443,E2 16828.443} C_VEL
LIN {X 0,Y 367.919,Z 1203,A -85,B 0,C 180,E1 16825.48,E2 16825.48} C_VEL
LIN {X 0,Y 368,Z 1201.246,A -85,B 0,C 180,E1 16822.349,E2 16822.349} C_VEL
LIN {X 0,Y 368.237,Z 1198.574,A -85,B 0,C 180,E1 16819.202,E2 16819.202} C_VEL
LIN {X 0,Y 368.815,Z 1194.766,A -85,B 0,C 180,E1 16815.878,E2 16815.878} C_VEL
LIN {X 0,Y 369.796,Z 1190.089,A -85,B 0,C 180,E1 16812.646,E2 16812.646} C_VEL
LIN {X 0,Y 371.399,Z 1184.292,A -85,B 0,C 180,E1 16809.349,E2 16809.349} C_VEL
LIN {X 0,Y 373.823,Z 1176.958,A -85,B 0,C 180,E1 16805.844,E2 16805.844} C_VEL
LIN {X 0,Y 378.028,Z 1166.231,A -85,B 0,C 180,E1 16801.57,E2 16801.57} C_VEL
LIN {X 0,Y 382.73,Z 1155.357,A -85,B 0,C 180,E1 16797.973,E2 16797.973} C_VEL
LIN {X 0,Y 387.758,Z 1144.624,A -85,B 0,C 180,E1 16794.899,E2 16794.899} C_VEL
LIN {X 0,Y 393.422,Z 1133.013,A -85,B 0,C 180,E1 16791.987,E2 16791.987} C_VEL
LIN {X 0,Y 401.375,Z 1117.313,A -85,B 0,C 180,E1 16788.577,E2 16788.577} C_VEL
LIN {X 0,Y 409.715,Z 1100.691,A -85,B 0,C 180,E1 16785.542,E2 16785.542} C_VEL
LIN {X 0,Y 417.049,Z 1086.016,A -85,B 0,C 180,E1 16783.212,E2 16783.212} C_VEL
LIN {X 0,Y 424.544,Z 1070.725,A -85,B 0,C 180,E1 16781.08,E2 16781.08} C_VEL
LIN {X 0,Y 432.156,Z 1054.698,A -85,B 0,C 180,E1 16779.116,E2 16779.116} C_VEL
LIN {X 0,Y 441.005,Z 1035.341,A -85,B 0,C 180,E1 16777.055,E2 16777.055} C_VEL
LIN {X 0,Y 450.864,Z 1012.17,A -85,B 0,C 180,E1 16774.973,E2 16774.973} C_VEL
LIN {X 0,Y 458.533,Z 992.719,A -85,B 0,C 180,E1 16773.484,E2 16773.484} C_VEL
LIN {X 0,Y 465.604,Z 973.446,A -85,B 0,C 180,E1 16772.211,E2 16772.211} C_VEL
LIN {X 0,Y 472.197,Z 953.78,A -85,B 0,C 180,E1 16771.085,E2 16771.085} C_VEL
LIN {X 0,Y 479.81,Z 928.671,A -85,B 0,C 180,E1 16769.872,E2 16769.872} C_VEL
LIN {X 0,Y 486.191,Z 903.735,A -85,B 0,C 180,E1 16768.901,E2 16768.901} C_VEL
LIN {X 0,Y 490.975,Z 882.004,A -85,B 0,C 180,E1 16768.205,E2 16768.205} C_VEL
LIN {X 0,Y 494.937,Z 860.701,A -85,B 0,C 180,E1 16767.652,E2 16767.652} C_VEL
LIN {X 0,Y 498.406,Z 837.411,A -85,B 0,C 180,E1 16767.171,E2 16767.171} C_VEL
LIN {X 0,Y 501.782,Z 801.462,A -85,B 0,C 180,E1 16766.568,E2 16766.568} C_VEL
LIN {X 0,Y 518.722,Z 580.856,A -85,B 0,C 180,E1 16763.135,E2 16763.135} C_VEL
LIN {X 0,Y 522.397,Z 534.048,A -85,B 0,C 180,E1 16762.389,E2 16762.389} C_VEL
LIN {X 0,Y 516.026,Z 523.053,A -85,B 0,C 180,E1 16759.763,E2 16759.763} C_VEL
LIN {X 0,Y 512.073,Z 517.162,A -85,B 0,C 180,E1 16757.911,E2 16757.911} C_VEL
LIN {X 0,Y 509.463,Z 513.32,A -85,B 0,C 180,E1 16756.534,E2 16756.534} C_VEL
LIN {X 0,Y 506.508,Z 508.899,A -85,B 0,C 180,E1 16754.753,E2 16754.753} C_VEL
LIN {X 0,Y 503.411,Z 504.369,A -85,B 0,C 180,E1 16752.504,E2 16752.504} C_VEL
LIN {X 0,Y 500.376,Z 499.801,A -85,B 0,C 180,E1 16749.489,E2 16749.489} C_VEL
LIN {X 0,Y 499.886,Z 499.107,A -85,B 0,C 180,E1 16748.855,E2 16748.855} C_VEL
LIN {X 0,Y 497.833,Z 497.141,A -85,B 0,C 180,E1 16743.916,E2 16743.916} C_VEL
LIN {X 0,Y 498.225,Z 497.703,A -85,B 0,C 180,E1 16740.92,E2 16740.92} C_VEL
LIN {X 0,Y 500.253,Z 499.472,A -85,B 0,C 180,E1 16737.48,E2 16737.48} C_VEL
LIN {X 0,Y 502.972,Z 503.951,A -85,B 0,C 180,E1 16734.639,E2 16734.639} C_VEL
LIN {X 0,Y 504.035,Z 505.275,A -85,B 0,C 180,E1 16733.793,E2 16733.793} C_VEL
LIN {X 0,Y 507.636,Z 510.51,A -85,B 0,C 180,E1 16731.333,E2 16731.333} C_VEL
LIN {X 0,Y 511.272,Z 515.939,A -85,B 0,C 180,E1 16729.293,E2 16729.293} C_VEL
LIN {X 0,Y 515.103,Z 521.664,A -85,B 0,C 180,E1 16727.443,E2 16727.443} C_VEL
LIN {X 0,Y 520.389,Z 529.737,A -85,B 0,C 180,E1 16725.222,E2 16725.222} C_VEL
LIN {X 0,Y 522.428,Z 533.029,A -85,B 0,C 180,E1 16724.437,E2 16724.437} C_VEL
LIN {X 0,Y 505.639,Z 748.197,A -85,B 0,C 180,E1 16721.093,E2 16721.093} C_VEL
LIN {X 0,Y 499.883,Z 821.492,A -85,B 0,C 180,E1 16719.935,E2 16719.935} C_VEL
LIN {X 0,Y 496.158,Z 850.239,A -85,B 0,C 180,E1 16719.379,E2 16719.379} C_VEL
LIN {X 0,Y 491.818,Z 874.467,A -85,B 0,C 180,E1 16718.762,E2 16718.762} C_VEL
LIN {X 0,Y 487.346,Z 895.313,A -85,B 0,C 180,E1 16718.102,E2 16718.102} C_VEL
LIN {X 0,Y 482.395,Z 915.26,A -85,B 0,C 180,E1 16717.348,E2 16717.348} C_VEL
LIN {X 0,Y 476.68,Z 935.638,A -85,B 0,C 180,E1 16716.438,E2 16716.438} C_VEL
LIN {X 0,Y 468.951,Z 960.222,A -85,B 0,C 180,E1 16715.137,E2 16715.137} C_VEL
LIN {X 0,Y 460.395,Z 983.895,A -85,B 0,C 180,E1 16713.616,E2 16713.616} C_VEL
LIN {X 0,Y 453.158,Z 1002.431,A -85,B 0,C 180,E1 16712.224,E2 16712.224} C_VEL
LIN {X 0,Y 445.887,Z 1019.851,A -85,B 0,C 180,E1 16710.726,E2 16710.726} C_VEL
LIN {X 0,Y 438.335,Z 1036.902,A -85,B 0,C 180,E1 16709.056,E2 16709.056} C_VEL
LIN {X 0,Y 429.032,Z 1056.966,A -85,B 0,C 180,E1 16706.788,E2 16706.788} C_VEL
LIN {X 0,Y 419.374,Z 1076.519,A -85,B 0,C 180,E1 16704.156,E2 16704.156} C_VEL
LIN {X 0,Y 411.735,Z 1091.614,A -85,B 0,C 180,E1 16701.803,E2 16701.803} C_VEL
LIN {X 0,Y 404.648,Z 1105.456,A -85,B 0,C 180,E1 16699.339,E2 16699.339} C_VEL
LIN {X 0,Y 397.018,Z 1120.394,A -85,B 0,C 180,E1 16696.285,E2 16696.285} C_VEL
LIN {X 0,Y 389.453,Z 1135.334,A -85,B 0,C 180,E1 16692.67,E2 16692.67} C_VEL
LIN {X 0,Y 383.932,Z 1146.688,A -85,B 0,C 180,E1 16689.452,E2 16689.452} C_VEL
LIN {X 0,Y 379.469,Z 1156.444,A -85,B 0,C 180,E1 16686.263,E2 16686.263} C_VEL
LIN {X 0,Y 375.563,Z 1165.802,A -85,B 0,C 180,E1 16682.714,E2 16682.714} C_VEL
LIN {X 0,Y 371.931,Z 1175.725,A -85,B 0,C 180,E1 16678.141,E2 16678.141} C_VEL
LIN {X 0,Y 370.069,Z 1181.964,A -85,B 0,C 180,E1 16674.587,E2 16674.587} C_VEL
LIN {X 0,Y 368.973,Z 1186.698,A -85,B 0,C 180,E1 16671.292,E2 16671.292} C_VEL
LIN {X 0,Y 368.333,Z 1190.415,A -85,B 0,C 180,E1 16668.027,E2 16668.027} C_VEL
LIN {X 0,Y 368.048,Z 1193.15,A -85,B 0,C 180,E1 16664.795,E2 16664.795} C_VEL
LIN {X 0,Y 367.936,Z 1194.864,A -85,B 0,C 180,E1 16661.76,E2 16661.76} C_VEL
LIN {X 0,Y 367.916,Z 1195.74,A -85,B 0,C 180,E1 16658.754,E2 16658.754} C_VEL
LIN {X 0,Y 367.917,Z 1195.795,A -85,B 0,C 180,E1 16655.771,E2 16655.771} C_VEL
LIN {X 0,Y 367.927,Z 1194.972,A -85,B 0,C 180,E1 16652.648,E2 16652.648} C_VEL
LIN {X 0,Y 368.021,Z 1193.258,A -85,B 0,C 180,E1 16649.533,E2 16649.533} C_VEL
LIN {X 0,Y 368.257,Z 1190.654,A -85,B 0,C 180,E1 16646.42,E2 16646.42} C_VEL
LIN {X 0,Y 368.812,Z 1186.946,A -85,B 0,C 180,E1 16643.149,E2 16643.149} C_VEL
LIN {X 0,Y 369.799,Z 1182.228,A -85,B 0,C 180,E1 16639.878,E2 16639.878} C_VEL
LIN {X 0,Y 371.361,Z 1176.471,A -85,B 0,C 180,E1 16636.612,E2 16636.612} C_VEL
LIN {X 0,Y 373.771,Z 1168.953,A -85,B 0,C 180,E1 16633.047,E2 16633.047} C_VEL
LIN {X 0,Y 375.545,Z 1164,A -85,B 0,C 180,E1 16631.026,E2 16631.026} C_VEL
LIN {X 0,Y 375.667,Z 1161.325,A -85,B 0,C 180,E1 16629.914,E2 16629.914} C_VEL
LIN {X 0,Y 372.904,Z 1154.208,A -85,B 0,C 180,E1 16626.876,E2 16626.876} C_VEL
LIN {X 0,Y 373.34,Z 1151.48,A -85,B 0,C 180,E1 16625.944,E2 16625.944} C_VEL
LIN {X 0,Y 379.103,Z 1138.676,A -85,B 0,C 180,E1 16622.172,E2 16622.172} C_VEL
LIN {X 0,Y 384.364,Z 1127.602,A -85,B 0,C 180,E1 16619.346,E2 16619.346} C_VEL
LIN {X 0,Y 390.33,Z 1115.254,A -85,B 0,C 180,E1 16616.583,E2 16616.583} C_VEL
LIN {X 0,Y 397.4,Z 1100.765,A -85,B 0,C 180,E1 16613.754,E2 16613.754} C_VEL
LIN {X 0,Y 406.686,Z 1081.334,A -85,B 0,C 180,E1 16610.535,E2 16610.535} C_VEL
LIN {X 0,Y 414.043,Z 1065.534,A -85,B 0,C 180,E1 16608.295,E2 16608.295} C_VEL
LIN {X 0,Y 421.481,Z 1049.039,A -85,B 0,C 180,E1 16606.25,E2 16606.25} C_VEL
LIN {X 0,Y 429.38,Z 1030.737,A -85,B 0,C 180,E1 16604.271,E2 16604.271} C_VEL
LIN {X 0,Y 439.041,Z 1006.675,A -85,B 0,C 180,E1 16602.062,E2 16602.062} C_VEL
LIN {X 0,Y 446.177,Z 987.425,A -85,B 0,C 180,E1 16600.564,E2 16600.564} C_VEL
LIN {X 0,Y 452.718,Z 968.375,A -85,B 0,C 180,E1 16599.277,E2 16599.277} C_VEL
LIN {X 0,Y 458.827,Z 948.841,A -85,B 0,C 180,E1 16598.124,E2 16598.124} C_VEL
LIN {X 0,Y 465.763,Z 924.413,A -85,B 0,C 180,E1 16596.904,E2 16596.904} C_VEL
LIN {X 0,Y 471.899,Z 898.707,A -85,B 0,C 180,E1 16595.861,E2 16595.861} C_VEL
LIN {X 0,Y 476.358,Z 876.961,A -85,B 0,C 180,E1 16595.141,E2 16595.141} C_VEL
LIN {X 0,Y 480,Z 855.726,A -85,B 0,C 180,E1 16594.562,E2 16594.562} C_VEL
LIN {X 0,Y 483.262,Z 832.119,A -85,B 0,C 180,E1 16594.056,E2 16594.056} C_VEL
LIN {X 0,Y 486.325,Z 796.3,A -85,B 0,C 180,E1 16593.451,E2 16593.451} C_VEL
LIN {X 0,Y 501.71,Z 572.725,A -85,B 0,C 180,E1 16589.967,E2 16589.967} C_VEL
LIN {X 0,Y 504.668,Z 530.54,A -85,B 0,C 180,E1 16589.3,E2 16589.3} C_VEL
LIN {X 0,Y 496.746,Z 518.171,A -85,B 0,C 180,E1 16586.833,E2 16586.833} C_VEL
LIN {X 0,Y 489.797,Z 507.678,A -85,B 0,C 180,E1 16584.386,E2 16584.386} C_VEL
LIN {X 0,Y 483.238,Z 498.219,A -85,B 0,C 180,E1 16581.739,E2 16581.739} C_VEL
LIN {X 0,Y 479.092,Z 492.528,A -85,B 0,C 180,E1 16579.825,E2 16579.825} C_VEL
LIN {X 0,Y 475.836,Z 487.928,A -85,B 0,C 180,E1 16578.119,E2 16578.119} C_VEL
LIN {X 0,Y 472.654,Z 483.516,A -85,B 0,C 180,E1 16576.215,E2 16576.215} C_VEL
LIN {X 0,Y 469.512,Z 479.299,A -85,B 0,C 180,E1 16573.988,E2 16573.988} C_VEL
LIN {X 0,Y 468.701,Z 478.148,A -85,B 0,C 180,E1 16573.321,E2 16573.321} C_VEL
LIN {X 0,Y 465.941,Z 474.734,A -85,B 0,C 180,E1 16570.635,E2 16570.635} C_VEL
LIN {X 0,Y 464.979,Z 472.679,A -85,B 0,C 180,E1 16569.281,E2 16569.281} C_VEL
LIN {X 0,Y 462.887,Z 471.241,A -85,B 0,C 180,E1 16563.84,E2 16563.84} C_VEL
LIN {X 0,Y 464.178,Z 472.247,A -85,B 0,C 180,E1 16559.013,E2 16559.013} C_VEL
LIN {X 0,Y 465.268,Z 473.085,A -85,B 0,C 180,E1 16557.413,E2 16557.413} C_VEL
LIN {X 0,Y 467.323,Z 476.873,A -85,B 0,C 180,E1 16554.967,E2 16554.967} C_VEL
LIN {X 0,Y 469.261,Z 478.785,A -85,B 0,C 180,E1 16553.331,E2 16553.331} C_VEL
LIN {X 0,Y 472.306,Z 483.114,A -85,B 0,C 180,E1 16551.11,E2 16551.11} C_VEL
LIN {X 0,Y 473.628,Z 484.834,A -85,B 0,C 180,E1 16550.277,E2 16550.277} C_VEL
LIN {X 0,Y 477.372,Z 490.07,A -85,B 0,C 180,E1 16548.155,E2 16548.155} C_VEL
LIN {X 0,Y 481.657,Z 496.062,A -85,B 0,C 180,E1 16546.066,E2 16546.066} C_VEL
LIN {X 0,Y 487.104,Z 503.707,A -85,B 0,C 180,E1 16543.759,E2 16543.759} C_VEL
LIN {X 0,Y 494.578,Z 514.769,A -85,B 0,C 180,E1 16541.004,E2 16541.004} C_VEL
LIN {X 0,Y 499.972,Z 523.805,A -85,B 0,C 180,E1 16539.208,E2 16539.208} C_VEL
LIN {X 0,Y 504.7,Z 532.127,A -85,B 0,C 180,E1 16537.744,E2 16537.744} C_VEL
LIN {X 0,Y 489.571,Z 749.986,A -85,B 0,C 180,E1 16534.349,E2 16534.349} C_VEL
LIN {X 0,Y 484.219,Z 826.081,A -85,B 0,C 180,E1 16533.141,E2 16533.141} C_VEL
LIN {X 0,Y 480.797,Z 854.575,A -85,B 0,C 180,E1 16532.588,E2 16532.588} C_VEL
LIN {X 0,Y 476.561,Z 879.576,A -85,B 0,C 180,E1 16531.948,E2 16531.948} C_VEL
LIN {X 0,Y 472.345,Z 900.467,A -85,B 0,C 180,E1 16531.28,E2 16531.28} C_VEL
LIN {X 0,Y 467.562,Z 920.923,A -85,B 0,C 180,E1 16530.499,E2 16530.499} C_VEL
LIN {X 0,Y 461.801,Z 942.7,A -85,B 0,C 180,E1 16529.51,E2 16529.51} C_VEL
LIN {X 0,Y 453.721,Z 969.482,A -85,B 0,C 180,E1 16528.04,E2 16528.04} C_VEL
LIN {X 0,Y 446.792,Z 989.917,A -85,B 0,C 180,E1 16526.703,E2 16526.703} C_VEL
LIN {X 0,Y 439.877,Z 1008.858,A -85,B 0,C 180,E1 16525.268,E2 16525.268} C_VEL
LIN {X 0,Y 432.893,Z 1026.745,A -85,B 0,C 180,E1 16523.715,E2 16523.715} C_VEL
LIN {X 0,Y 424.691,Z 1046.563,A -85,B 0,C 180,E1 16521.742,E2 16521.742} C_VEL
LIN {X 0,Y 415.233,Z 1067.941,A -85,B 0,C 180,E1 16519.226,E2 16519.226} C_VEL
LIN {X 0,Y 407.876,Z 1083.93,A -85,B 0,C 180,E1 16517.038,E2 16517.038} C_VEL
LIN {X 0,Y 401.241,Z 1098.034,A -85,B 0,C 180,E1 16514.846,E2 16514.846} C_VEL
LIN {X 0,Y 394.578,Z 1112.021,A -85,B 0,C 180,E1 16512.38,E2 16512.38} C_VEL
LIN {X 0,Y 387.199,Z 1127.514,A -85,B 0,C 180,E1 16509.246,E2 16509.246} C_VEL
LIN {X 0,Y 380.053,Z 1142.632,A -85,B 0,C 180,E1 16505.614,E2 16505.614} C_VEL
LIN {X 0,Y 374.889,Z 1154.034,A -85,B 0,C 180,E1 16502.417,E2 16502.417} C_VEL
LIN {X 0,Y 370.67,Z 1163.924,A -85,B 0,C 180,E1 16499.225,E2 16499.225} C_VEL
LIN {X 0,Y 366.847,Z 1173.821,A -85,B 0,C 180,E1 16495.508,E2 16495.508} C_VEL
LIN {X 0,Y 363.602,Z 1183.387,A -85,B 0,C 180,E1 16491.114,E2 16491.114} C_VEL
LIN {X 0,Y 361.847,Z 1189.681,A -85,B 0,C 180,E1 16487.571,E2 16487.571} C_VEL
LIN {X 0,Y 360.838,Z 1194.47,A -85,B 0,C 180,E1 16484.277,E2 16484.277} C_VEL
LIN {X 0,Y 360.257,Z 1198.206,A -85,B 0,C 180,E1 16481.04,E2 16481.04} C_VEL
LIN {X 0,Y 360.005,Z 1200.979,A -85,B 0,C 180,E1 16477.822,E2 16477.822} C_VEL
LIN {X 0,Y 359.925,Z 1202.744,A -85,B 0,C 180,E1 16474.78,E2 16474.78} C_VEL
LIN {X 0,Y 359.912,Z 1203.676,A -85,B 0,C 180,E1 16471.751,E2 16471.751} C_VEL
LIN {X 0,Y 359.915,Z 1203.782,A -85,B 0,C 180,E1 16468.727,E2 16468.727} C_VEL
LIN {X 0,Y 359.919,Z 1202.996,A -85,B 0,C 180,E1 16465.539,E2 16465.539} C_VEL
LIN {X 0,Y 360.001,Z 1201.299,A -85,B 0,C 180,E1 16462.339,E2 16462.339} C_VEL
LIN {X 0,Y 360.263,Z 1198.526,A -85,B 0,C 180,E1 16458.96,E2 16458.96} C_VEL
LIN {X 0,Y 360.894,Z 1194.731,A -85,B 0,C 180,E1 16455.561,E2 16455.561} C_VEL
LIN {X 0,Y 361.93,Z 1190.147,A -85,B 0,C 180,E1 16452.309,E2 16452.309} C_VEL
LIN {X 0,Y 363.663,Z 1184.288,A -85,B 0,C 180,E1 16448.889,E2 16448.889} C_VEL
LIN {X 0,Y 366.253,Z 1176.971,A -85,B 0,C 180,E1 16445.312,E2 16445.312} C_VEL
LIN {X 0,Y 370.745,Z 1166.15,A -85,B 0,C 180,E1 16440.906,E2 16440.906} C_VEL
LIN {X 0,Y 375.906,Z 1154.92,A -85,B 0,C 180,E1 16437.138,E2 16437.138} C_VEL
LIN {X 0,Y 381.197,Z 1144.159,A -85,B 0,C 180,E1 16434.018,E2 16434.018} C_VEL
LIN {X 0,Y 387.741,Z 1131.451,A -85,B 0,C 180,E1 16430.819,E2 16430.819} C_VEL
LIN {X 0,Y 396.851,Z 1114.172,A -85,B 0,C 180,E1 16427.136,E2 16427.136} C_VEL
LIN {X 0,Y 404.672,Z 1099.238,A -85,B 0,C 180,E1 16424.434,E2 16424.434} C_VEL
LIN {X 0,Y 412.35,Z 1084.441,A -85,B 0,C 180,E1 16422.1,E2 16422.1} C_VEL
LIN {X 0,Y 420.136,Z 1069.08,A -85,B 0,C 180,E1 16419.977,E2 16419.977} C_VEL
LIN {X 0,Y 428.988,Z 1051.031,A -85,B 0,C 180,E1 16417.803,E2 16417.803} C_VEL
LIN {X 0,Y 439.545,Z 1028.112,A -85,B 0,C 180,E1 16415.476,E2 16415.476} C_VEL
LIN {X 0,Y 447.455,Z 1009.76,A -85,B 0,C 180,E1 16413.888,E2 16413.888} C_VEL
LIN {X 0,Y 455.058,Z 990.853,A -85,B 0,C 180,E1 16412.464,E2 16412.464} C_VEL
LIN {X 0,Y 462.635,Z 970.519,A -85,B 0,C 180,E1 16411.147,E2 16411.147} C_VEL
LIN {X 0,Y 471.123,Z 945.297,A -85,B 0,C 180,E1 16409.772,E2 16409.772} C_VEL
LIN {X 0,Y 477.818,Z 922.362,A -85,B 0,C 180,E1 16408.744,E2 16408.744} C_VEL
LIN {X 0,Y 483.298,Z 901.039,A -85,B 0,C 180,E1 16407.947,E2 16407.947} C_VEL
LIN {X 0,Y 487.997,Z 879.842,A -85,B 0,C 180,E1 16407.289,E2 16407.289} C_VEL
LIN {X 0,Y 492.246,Z 857.016,A -85,B 0,C 180,E1 16406.719,E2 16406.719} C_VEL
LIN {X 0,Y 496.388,Z 826.742,A -85,B 0,C 180,E1 16406.135,E2 16406.135} C_VEL
LIN {X 0,Y 501.522,Z 763.434,A -85,B 0,C 180,E1 16405.131,E2 16405.131} C_VEL
LIN {X 0,Y 519.118,Z 542.765,A -85,B 0,C 180,E1 16401.709,E2 16401.709} C_VEL
LIN {X 0,Y 519.333,Z 539.365,A -85,B 0,C 180,E1 16401.636,E2 16401.636} C_VEL
LIN {X 0,Y 514.07,Z 530.06,A -85,B 0,C 180,E1 16399.368,E2 16399.368} C_VEL
LIN {X 0,Y 508.904,Z 522.028,A -85,B 0,C 180,E1 16396.788,E2 16396.788} C_VEL
LIN {X 0,Y 505.189,Z 516.609,A -85,B 0,C 180,E1 16394.558,E2 16394.558} C_VEL
LIN {X 0,Y 502.158,Z 512.12,A -85,B 0,C 180,E1 16392.302,E2 16392.302} C_VEL
LIN {X 0,Y 499.225,Z 507.505,A -85,B 0,C 180,E1 16389.278,E2 16389.278} C_VEL
LIN {X 0,Y 496.962,Z 505.207,A -85,B 0,C 180,E1 16384.732,E2 16384.732} C_VEL
LIN {X 0,Y 497.007,Z 505.247,A -85,B 0,C 180,E1 16381.845,E2 16381.845} C_VEL
LIN {X 0,Y 499.175,Z 507.375,A -85,B 0,C 180,E1 16377.589,E2 16377.589} C_VEL
LIN {X 0,Y 501.851,Z 511.821,A -85,B 0,C 180,E1 16374.741,E2 16374.741} C_VEL
LIN {X 0,Y 502.891,Z 513.215,A -85,B 0,C 180,E1 16373.894,E2 16373.894} C_VEL
LIN {X 0,Y 506.274,Z 518.189,A -85,B 0,C 180,E1 16371.539,E2 16371.539} C_VEL
LIN {X 0,Y 509.843,Z 523.629,A -85,B 0,C 180,E1 16369.491,E2 16369.491} C_VEL
LIN {X 0,Y 513.734,Z 529.539,A -85,B 0,C 180,E1 16367.58,E2 16367.58} C_VEL
LIN {X 0,Y 519.161,Z 538.027,A -85,B 0,C 180,E1 16365.272,E2 16365.272} C_VEL
LIN {X 0,Y 519.336,Z 538.698,A -85,B 0,C 180,E1 16365.186,E2 16365.186} C_VEL
LIN {X 0,Y 502.227,Z 752.631,A -85,B 0,C 180,E1 16361.869,E2 16361.869} C_VEL
LIN {X 0,Y 496.638,Z 821.759,A -85,B 0,C 180,E1 16360.777,E2 16360.777} C_VEL
LIN {X 0,Y 492.752,Z 850.907,A -85,B 0,C 180,E1 16360.215,E2 16360.215} C_VEL
LIN {X 0,Y 488.378,Z 874.773,A -85,B 0,C 180,E1 16359.61,E2 16359.61} C_VEL
LIN {X 0,Y 483.896,Z 895.238,A -85,B 0,C 180,E1 16358.968,E2 16358.968} C_VEL
LIN {X 0,Y 478.841,Z 915.203,A -85,B 0,C 180,E1 16358.22,E2 16358.22} C_VEL
LIN {X 0,Y 473.012,Z 935.531,A -85,B 0,C 180,E1 16357.32,E2 16357.32} C_VEL
LIN {X 0,Y 465.37,Z 959.299,A -85,B 0,C 180,E1 16356.076,E2 16356.076} C_VEL
LIN {X 0,Y 456.335,Z 983.819,A -85,B 0,C 180,E1 16354.517,E2 16354.517} C_VEL
LIN {X 0,Y 448.59,Z 1003.126,A -85,B 0,C 180,E1 16353.069,E2 16353.069} C_VEL
LIN {X 0,Y 441.125,Z 1020.476,A -85,B 0,C 180,E1 16351.575,E2 16351.575} C_VEL
LIN {X 0,Y 432.784,Z 1038.734,A -85,B 0,C 180,E1 16349.774,E2 16349.774} C_VEL
LIN {X 0,Y 422.146,Z 1060.652,A -85,B 0,C 180,E1 16347.227,E2 16347.227} C_VEL
LIN {X 0,Y 413.574,Z 1077.412,A -85,B 0,C 180,E1 16344.927,E2 16344.927} C_VEL
LIN {X 0,Y 406.081,Z 1091.689,A -85,B 0,C 180,E1 16342.683,E2 16342.683} C_VEL
LIN {X 0,Y 398.896,Z 1105.175,A -85,B 0,C 180,E1 16340.268,E2 16340.268} C_VEL
LIN {X 0,Y 391.738,Z 1118.559,A -85,B 0,C 180,E1 16337.53,E2 16337.53} C_VEL
LIN {X 0,Y 383.335,Z 1134.436,A -85,B 0,C 180,E1 16333.725,E2 16333.725} C_VEL
LIN {X 0,Y 377.195,Z 1146.416,A -85,B 0,C 180,E1 16330.3,E2 16330.3} C_VEL
LIN {X 0,Y 372.557,Z 1155.971,A -85,B 0,C 180,E1 16327.145,E2 16327.145} C_VEL
LIN {X 0,Y 368.593,Z 1164.77,A -85,B 0,C 180,E1 16323.786,E2 16323.786} C_VEL
LIN {X 0,Y 365.02,Z 1173.815,A -85,B 0,C 180,E1 16319.722,E2 16319.722} C_VEL
LIN {X 0,Y 362.409,Z 1181.609,A -85,B 0,C 180,E1 16315.317,E2 16315.317} C_VEL
LIN {X 0,Y 361.11,Z 1186.638,A -85,B 0,C 180,E1 16311.779,E2 16311.779} C_VEL
LIN {X 0,Y 360.391,Z 1190.424,A -85,B 0,C 180,E1 16308.401,E2 16308.401} C_VEL
LIN {X 0,Y 360.073,Z 1193.155,A -85,B 0,C 180,E1 16305.131,E2 16305.131} C_VEL
LIN {X 0,Y 359.943,Z 1194.903,A -85,B 0,C 180,E1 16302.025,E2 16302.025} C_VEL
LIN {X 0,Y 359.917,Z 1195.812,A -85,B 0,C 180,E1 16298.95,E2 16298.95} C_VEL
LIN {X 0,Y 359.918,Z 1195.899,A -85,B 0,C 180,E1 16295.9,E2 16295.9} C_VEL
LIN {X 0,Y 359.927,Z 1195.109,A -85,B 0,C 180,E1 16292.707,E2 16292.707} C_VEL
LIN {X 0,Y 360.023,Z 1193.428,A -85,B 0,C 180,E1 16289.523,E2 16289.523} C_VEL
LIN {X 0,Y 360.286,Z 1190.699,A -85,B 0,C 180,E1 16286.181,E2 16286.181} C_VEL
LIN {X 0,Y 360.892,Z 1186.978,A -85,B 0,C 180,E1 16282.838,E2 16282.838} C_VEL
LIN {X 0,Y 361.952,Z 1182.246,A -85,B 0,C 180,E1 16279.495,E2 16279.495} C_VEL
LIN {X 0,Y 363.715,Z 1176.18,A -85,B 0,C 180,E1 16276.001,E2 16276.001} C_VEL
LIN {X 0,Y 366.868,Z 1167.174,A -85,B 0,C 180,E1 16271.735,E2 16271.735} C_VEL
LIN {X 0,Y 370.906,Z 1156.958,A -85,B 0,C 180,E1 16267.827,E2 16267.827} C_VEL
LIN {X 0,Y 373.34,Z 1151.48,A -85,B 0,C 180,E1 16265.944,E2 16265.944} C_VEL
LIN {X 0,Y 373.819,Z 1148.262,A -85,B 0,C 180,E1 16264.865,E2 16264.865} C_VEL
LIN {X 0,Y 372.216,Z 1140.425,A -85,B 0,C 180,E1 16262.029,E2 16262.029} C_VEL
LIN {X 0,Y 373.056,Z 1136.873,A -85,B 0,C 180,E1 16260.969,E2 16260.969} C_VEL
LIN {X 0,Y 379.91,Z 1123.163,A -85,B 0,C 180,E1 16257.528,E2 16257.528} C_VEL
LIN {X 0,Y 388.257,Z 1106.576,A -85,B 0,C 180,E1 16254.045,E2 16254.045} C_VEL
LIN {X 0,Y 395.257,Z 1092.588,A -85,B 0,C 180,E1 16251.517,E2 16251.517} C_VEL
LIN {X 0,Y 402.451,Z 1077.974,A -85,B 0,C 180,E1 16249.202,E2 16249.202} C_VEL
LIN {X 0,Y 410.191,Z 1061.804,A -85,B 0,C 180,E1 16246.96,E2 16246.96} C_VEL
LIN {X 0,Y 420.226,Z 1039.891,A -85,B 0,C 180,E1 16244.368,E2 16244.368} C_VEL
LIN {X 0,Y 428.325,Z 1020.938,A -85,B 0,C 180,E1 16242.468,E2 16242.468} C_VEL
LIN {X 0,Y 435.402,Z 1003.341,A -85,B 0,C 180,E1 16240.93,E2 16240.93} C_VEL
LIN {X 0,Y 442.474,Z 984.521,A -85,B 0,C 180,E1 16239.495,E2 16239.495} C_VEL
LIN {X 0,Y 450.113,Z 962.51,A -85,B 0,C 180,E1 16238.051,E2 16238.051} C_VEL
LIN {X 0,Y 457.968,Z 936.789,A -85,B 0,C 180,E1 16236.646,E2 16236.646} C_VEL
LIN {X 0,Y 463.554,Z 916.076,A -85,B 0,C 180,E1 16235.7,E2 16235.7} C_VEL
LIN {X 0,Y 468.475,Z 895.367,A -85,B 0,C 180,E1 16234.9,E2 16234.9} C_VEL
LIN {X 0,Y 472.95,Z 873.464,A -85,B 0,C 180,E1 16234.197,E2 16234.197} C_VEL
LIN {X 0,Y 477.492,Z 846.48,A -85,B 0,C 180,E1 16233.51,E2 16233.51} C_VEL
LIN {X 0,Y 480.613,Z 819.753,A -85,B 0,C 180,E1 16233.002,E2 16233.002} C_VEL
LIN {X 0,Y 490.874,Z 675.588,A -85,B 0,C 180,E1 16230.735,E2 16230.735} C_VEL
LIN {X 0,Y 500.909,Z 535.275,A -85,B 0,C 180,E1 16228.531,E2 16228.531} C_VEL
LIN {X 0,Y 492.911,Z 522.692,A -85,B 0,C 180,E1 16225.922,E2 16225.922} C_VEL
LIN {X 0,Y 486.465,Z 512.989,A -85,B 0,C 180,E1 16223.536,E2 16223.536} C_VEL
LIN {X 0,Y 480.955,Z 504.936,A -85,B 0,C 180,E1 16221.207,E2 16221.207} C_VEL
LIN {X 0,Y 477.295,Z 499.78,A -85,B 0,C 180,E1 16219.457,E2 16219.457} C_VEL
LIN {X 0,Y 474.442,Z 495.631,A -85,B 0,C 180,E1 16217.921,E2 16217.921} C_VEL
LIN {X 0,Y 471.311,Z 491.236,A -85,B 0,C 180,E1 16216.01,E2 16216.01} C_VEL
LIN {X 0,Y 468.167,Z 486.864,A -85,B 0,C 180,E1 16213.714,E2 16213.714} C_VEL
LIN {X 0,Y 466.999,Z 485.553,A -85,B 0,C 180,E1 16212.74,E2 16212.74} C_VEL
LIN {X 0,Y 464.458,Z 481.714,A -85,B 0,C 180,E1 16209.98,E2 16209.98} C_VEL
LIN {X 0,Y 463.919,Z 480.587,A -85,B 0,C 180,E1 16209.178,E2 16209.178} C_VEL
LIN {X 0,Y 461.911,Z 479.182,A -85,B 0,C 180,E1 16203.848,E2 16203.848} C_VEL
LIN {X 0,Y 463.199,Z 480.193,A -85,B 0,C 180,E1 16199.011,E2 16199.011} C_VEL
LIN {X 0,Y 464.19,Z 480.996,A -85,B 0,C 180,E1 16197.531,E2 16197.531} C_VEL
LIN {X 0,Y 466.339,Z 484.886,A -85,B 0,C 180,E1 16194.957,E2 16194.957} C_VEL
LIN {X 0,Y 468.044,Z 486.603,A -85,B 0,C 180,E1 16193.499,E2 16193.499} C_VEL
LIN {X 0,Y 471.135,Z 490.994,A -85,B 0,C 180,E1 16191.21,E2 16191.21} C_VEL
LIN {X 0,Y 472.62,Z 493.137,A -85,B 0,C 180,E1 16190.256,E2 16190.256} C_VEL
LIN {X 0,Y 475.925,Z 497.771,A -85,B 0,C 180,E1 16188.364,E2 16188.364} C_VEL
LIN {X 0,Y 480.024,Z 503.59,A -85,B 0,C 180,E1 16186.325,E2 16186.325} C_VEL
LIN {X 0,Y 485.451,Z 511.396,A -85,B 0,C 180,E1 16183.978,E2 16183.978} C_VEL
LIN {X 0,Y 492.52,Z 522.004,A -85,B 0,C 180,E1 16181.321,E2 16181.321} C_VEL
LIN {X 0,Y 498.497,Z 532.226,A -85,B 0,C 180,E1 16179.297,E2 16179.297} C_VEL
LIN {X 0,Y 500.977,Z 536.893,A -85,B 0,C 180,E1 16178.5,E2 16178.5} C_VEL
LIN {X 0,Y 485.402,Z 755.448,A -85,B 0,C 180,E1 16175.095,E2 16175.095} C_VEL
LIN {X 0,Y 480.267,Z 826.313,A -85,B 0,C 180,E1 16173.969,E2 16173.969} C_VEL
LIN {X 0,Y 476.684,Z 855.22,A -85,B 0,C 180,E1 16173.406,E2 16173.406} C_VEL
LIN {X 0,Y 472.455,Z 879.633,A -85,B 0,C 180,E1 16172.783,E2 16172.783} C_VEL
LIN {X 0,Y 468.08,Z 900.815,A -85,B 0,C 180,E1 16172.107,E2 16172.107} C_VEL
LIN {X 0,Y 463.055,Z 921.775,A -85,B 0,C 180,E1 16171.306,E2 16171.306} C_VEL
LIN {X 0,Y 456.332,Z 946.479,A -85,B 0,C 180,E1 16170.172,E2 16170.172} C_VEL
LIN {X 0,Y 448.747,Z 970.528,A -85,B 0,C 180,E1 16168.825,E2 16168.825} C_VEL
LIN {X 0,Y 441.663,Z 990.851,A -85,B 0,C 180,E1 16167.488,E2 16167.488} C_VEL
LIN {X 0,Y 434.698,Z 1009.404,A -85,B 0,C 180,E1 16166.074,E2 16166.074} C_VEL
LIN {X 0,Y 427.146,Z 1028.186,A -85,B 0,C 180,E1 16164.431,E2 16164.431} C_VEL
LIN {X 0,Y 417.403,Z 1050.801,A -85,B 0,C 180,E1 16162.119,E2 16162.119} C_VEL
LIN {X 0,Y 408.903,Z 1069.295,A -85,B 0,C 180,E1 16159.88,E2 16159.88} C_VEL
LIN {X 0,Y 401.465,Z 1084.946,A -85,B 0,C 180,E1 16157.704,E2 16157.704} C_VEL
LIN {X 0,Y 394.314,Z 1099.617,A -85,B 0,C 180,E1 16155.379,E2 16155.379} C_VEL
LIN {X 0,Y 386.071,Z 1116.376,A -85,B 0,C 180,E1 16152.326,E2 16152.326} C_VEL
LIN {X 0,Y 378.327,Z 1131.849,A -85,B 0,C 180,E1 16148.976,E2 16148.976} C_VEL
LIN {X 0,Y 372.264,Z 1144.303,A -85,B 0,C 180,E1 16145.84,E2 16145.84} C_VEL
LIN {X 0,Y 367.173,Z 1155.133,A -85,B 0,C 180,E1 16142.704,E2 16142.704} C_VEL
LIN {X 0,Y 362.024,Z 1166.962,A -85,B 0,C 180,E1 16138.722,E2 16138.722} C_VEL
LIN {X 0,Y 358.006,Z 1176.999,A -85,B 0,C 180,E1 16134.591,E2 16134.591} C_VEL
LIN {X 0,Y 355.568,Z 1184.133,A -85,B 0,C 180,E1 16131.096,E2 16131.096} C_VEL
LIN {X 0,Y 353.848,Z 1190.103,A -85,B 0,C 180,E1 16127.599,E2 16127.599} C_VEL
LIN {X 0,Y 352.829,Z 1194.767,A -85,B 0,C 180,E1 16124.256,E2 16124.256} C_VEL
LIN {X 0,Y 352.23,Z 1198.561,A -85,B 0,C 180,E1 16120.798,E2 16120.798} C_VEL
LIN {X 0,Y 351.979,Z 1201.438,A -85,B 0,C 180,E1 16117.18,E2 16117.18} C_VEL
LIN {X 0,Y 351.916,Z 1203.391,A -85,B 0,C 180,E1 16113.094,E2 16113.094} C_VEL
LIN {X 0,Y 351.909,Z 1203.769,A -85,B 0,C 180,E1 16109.186,E2 16109.186} C_VEL
LIN {X 0,Y 351.918,Z 1202.995,A -85,B 0,C 180,E1 16105.6,E2 16105.6} C_VEL
LIN {X 0,Y 352.006,Z 1201.241,A -85,B 0,C 180,E1 16102.164,E2 16102.164} C_VEL
LIN {X 0,Y 352.292,Z 1198.479,A -85,B 0,C 180,E1 16098.707,E2 16098.707} C_VEL
LIN {X 0,Y 352.977,Z 1194.698,A -85,B 0,C 180,E1 16095.23,E2 16095.23} C_VEL
LIN {X 0,Y 354.172,Z 1189.876,A -85,B 0,C 180,E1 16091.738,E2 16091.738} C_VEL
LIN {X 0,Y 356.053,Z 1183.983,A -85,B 0,C 180,E1 16088.243,E2 16088.243} C_VEL
LIN {X 0,Y 359.004,Z 1176.286,A -85,B 0,C 180,E1 16084.425,E2 16084.425} C_VEL
LIN {X 0,Y 364.007,Z 1164.974,A -85,B 0,C 180,E1 16079.824,E2 16079.824} C_VEL
LIN {X 0,Y 369.142,Z 1154.492,A -85,B 0,C 180,E1 16076.271,E2 16076.271} C_VEL
LIN {X 0,Y 374.736,Z 1143.697,A -85,B 0,C 180,E1 16073.106,E2 16073.106} C_VEL
LIN {X 0,Y 381.648,Z 1130.957,A -85,B 0,C 180,E1 16069.873,E2 16069.873} C_VEL
LIN {X 0,Y 391.323,Z 1113.312,A -85,B 0,C 180,E1 16066.1,E2 16066.1} C_VEL
LIN {X 0,Y 399.326,Z 1098.626,A -85,B 0,C 180,E1 16063.438,E2 16063.438} C_VEL
LIN {X 0,Y 407.485,Z 1083.459,A -85,B 0,C 180,E1 16061.047,E2 16061.047} C_VEL
LIN {X 0,Y 416.201,Z 1066.833,A -85,B 0,C 180,E1 16058.77,E2 16058.77} C_VEL
LIN {X 0,Y 427.334,Z 1044.477,A -85,B 0,C 180,E1 16056.175,E2 16056.175} C_VEL
LIN {X 0,Y 436.177,Z 1025.583,A -85,B 0,C 180,E1 16054.328,E2 16054.328} C_VEL
LIN {X 0,Y 443.902,Z 1008.075,A -85,B 0,C 180,E1 16052.844,E2 16052.844} C_VEL
LIN {X 0,Y 451.416,Z 989.807,A -85,B 0,C 180,E1 16051.488,E2 16051.488} C_VEL
LIN {X 0,Y 459.518,Z 968.494,A -85,B 0,C 180,E1 16050.128,E2 16050.128} C_VEL
LIN {X 0,Y 468.213,Z 942.777,A -85,B 0,C 180,E1 16048.764,E2 16048.764} C_VEL
LIN {X 0,Y 474.735,Z 920.771,A -85,B 0,C 180,E1 16047.801,E2 16047.801} C_VEL
LIN {X 0,Y 480.161,Z 899.955,A -85,B 0,C 180,E1 16047.037,E2 16047.037} C_VEL
LIN {X 0,Y 485.035,Z 878.275,A -85,B 0,C 180,E1 16046.379,E2 16046.379} C_VEL
LIN {X 0,Y 489.987,Z 851.648,A -85,B 0,C 180,E1 16045.738,E2 16045.738} C_VEL
LIN {X 0,Y 493.497,Z 824.388,A -85,B 0,C 180,E1 16045.238,E2 16045.238} C_VEL
LIN {X 0,Y 505.855,Z 672.188,A -85,B 0,C 180,E1 16042.861,E2 16042.861} C_VEL
LIN {X 0,Y 516.369,Z 544.632,A -85,B 0,C 180,E1 16040.873,E2 16040.873} C_VEL
LIN {X 0,Y 512.254,Z 537.273,A -85,B 0,C 180,E1 16039.025,E2 16039.025} C_VEL
LIN {X 0,Y 507.423,Z 529.607,A -85,B 0,C 180,E1 16036.543,E2 16036.543} C_VEL
LIN {X 0,Y 503.876,Z 524.32,A -85,B 0,C 180,E1 16034.362,E2 16034.362} C_VEL
LIN {X 0,Y 500.911,Z 519.867,A -85,B 0,C 180,E1 16032.099,E2 16032.099} C_VEL
LIN {X 0,Y 498.081,Z 515.209,A -85,B 0,C 180,E1 16029.067,E2 16029.067} C_VEL
LIN {X 0,Y 495.9,Z 513.062,A -85,B 0,C 180,E1 16024.163,E2 16024.163} C_VEL
LIN {X 0,Y 496.161,Z 513.447,A -85,B 0,C 180,E1 16021.27,E2 16021.27} C_VEL
LIN {X 0,Y 498.099,Z 515.275,A -85,B 0,C 180,E1 16017.699,E2 16017.699} C_VEL
LIN {X 0,Y 500.867,Z 519.83,A -85,B 0,C 180,E1 16014.731,E2 16014.731} C_VEL
LIN {X 0,Y 501.957,Z 521.533,A -85,B 0,C 180,E1 16013.825,E2 16013.825} C_VEL
LIN {X 0,Y 504.92,Z 525.867,A -85,B 0,C 180,E1 16011.745,E2 16011.745} C_VEL
LIN {X 0,Y 508.421,Z 531.316,A -85,B 0,C 180,E1 16009.69,E2 16009.69} C_VEL
LIN {X 0,Y 513.088,Z 538.417,A -85,B 0,C 180,E1 16007.393,E2 16007.393} C_VEL
LIN {X 0,Y 516.374,Z 543.94,A -85,B 0,C 180,E1 16005.951,E2 16005.951} C_VEL
LIN {X 0,Y 498.875,Z 757.484,A -85,B 0,C 180,E1 16002.648,E2 16002.648} C_VEL
LIN {X 0,Y 493.492,Z 822.169,A -85,B 0,C 180,E1 16001.628,E2 16001.628} C_VEL
LIN {X 0,Y 489.387,Z 851.976,A -85,B 0,C 180,E1 16001.053,E2 16001.053} C_VEL
LIN {X 0,Y 485.035,Z 875.176,A -85,B 0,C 180,E1 16000.468,E2 16000.468} C_VEL
LIN {X 0,Y 480.412,Z 895.794,A -85,B 0,C 180,E1 15999.825,E2 15999.825} C_VEL
LIN {X 0,Y 475.05,Z 916.423,A -85,B 0,C 180,E1 15999.054,E2 15999.054} C_VEL
LIN {X 0,Y 468.394,Z 938.944,A -85,B 0,C 180,E1 15998.049,E2 15998.049} C_VEL
LIN {X 0,Y 459.582,Z 964.829,A -85,B 0,C 180,E1 15996.649,E2 15996.649} C_VEL
LIN {X 0,Y 451.716,Z 985.431,A -85,B 0,C 180,E1 15995.316,E2 15995.316} C_VEL
LIN {X 0,Y 444.123,Z 1003.824,A -85,B 0,C 180,E1 15993.932,E2 15993.932} C_VEL
LIN {X 0,Y 436.152,Z 1021.805,A -85,B 0,C 180,E1 15992.379,E2 15992.379} C_VEL
LIN {X 0,Y 426.128,Z 1043.075,A -85,B 0,C 180,E1 15990.245,E2 15990.245} C_VEL
LIN {X 0,Y 416.32,Z 1062.309,A -85,B 0,C 180,E1 15987.941,E2 15987.941} C_VEL
LIN {X 0,Y 408.083,Z 1077.881,A -85,B 0,C 180,E1 15985.783,E2 15985.783} C_VEL
LIN {X 0,Y 400.322,Z 1092.135,A -85,B 0,C 180,E1 15983.526,E2 15983.526} C_VEL
LIN {X 0,Y 392.539,Z 1106.196,A -85,B 0,C 180,E1 15980.976,E2 15980.976} C_VEL
LIN {X 0,Y 383.906,Z 1121.793,A -85,B 0,C 180,E1 15977.702,E2 15977.702} C_VEL
LIN {X 0,Y 375.692,Z 1136.497,A -85,B 0,C 180,E1 15973.997,E2 15973.997} C_VEL
LIN {X 0,Y 369.922,Z 1147.308,A -85,B 0,C 180,E1 15970.814,E2 15970.814} C_VEL
LIN {X 0,Y 364.917,Z 1157.152,A -85,B 0,C 180,E1 15967.465,E2 15967.465} C_VEL
LIN {X 0,Y 359.974,Z 1167.873,A -85,B 0,C 180,E1 15963.174,E2 15963.174} C_VEL
LIN {X 0,Y 356.395,Z 1176.536,A -85,B 0,C 180,E1 15958.851,E2 15958.851} C_VEL
LIN {X 0,Y 354.445,Z 1182.295,A -85,B 0,C 180,E1 15955.39,E2 15955.39} C_VEL
LIN {X 0,Y 353.163,Z 1186.998,A -85,B 0,C 180,E1 15951.945,E2 15951.945} C_VEL
LIN {X 0,Y 352.414,Z 1190.685,A -85,B 0,C 180,E1 15948.528,E2 15948.528} C_VEL
LIN {X 0,Y 352.086,Z 1193.278,A -85,B 0,C 180,E1 15945.314,E2 15945.314} C_VEL
LIN {X 0,Y 351.948,Z 1195.011,A -85,B 0,C 180,E1 15942.136,E2 15942.136} C_VEL
LIN {X 0,Y 351.917,Z 1195.906,A -85,B 0,C 180,E1 15938.99,E2 15938.99} C_VEL
LIN {X 0,Y 351.919,Z 1195.98,A -85,B 0,C 180,E1 15935.871,E2 15935.871} C_VEL
LIN {X 0,Y 351.928,Z 1195.177,A -85,B 0,C 180,E1 15932.605,E2 15932.605} C_VEL
LIN {X 0,Y 352.027,Z 1193.483,A -85,B 0,C 180,E1 15929.349,E2 15929.349} C_VEL
LIN {X 0,Y 352.299,Z 1190.898,A -85,B 0,C 180,E1 15926.094,E2 15926.094} C_VEL
LIN {X 0,Y 352.936,Z 1187.209,A -85,B 0,C 180,E1 15922.676,E2 15922.676} C_VEL
LIN {X 0,Y 354.048,Z 1182.509,A -85,B 0,C 180,E1 15919.258,E2 15919.258} C_VEL
LIN {X 0,Y 355.816,Z 1176.704,A -85,B 0,C 180,E1 15915.813,E2 15915.813} C_VEL
LIN {X 0,Y 358.481,Z 1169.267,A -85,B 0,C 180,E1 15912.133,E2 15912.133} C_VEL
LIN {X 0,Y 363.036,Z 1158.242,A -85,B 0,C 180,E1 15907.662,E2 15907.662} C_VEL
LIN {X 0,Y 367.799,Z 1147.782,A -85,B 0,C 180,E1 15904.139,E2 15904.139} C_VEL
LIN {X 0,Y 373.039,Z 1136.908,A -85,B 0,C 180,E1 15900.979,E2 15900.979} C_VEL
LIN {X 0,Y 373.056,Z 1136.873,A -85,B 0,C 180,E1 15900.969,E2 15900.969} C_VEL
LIN {X 0,Y 373.981,Z 1133.362,A -85,B 0,C 180,E1 15899.918,E2 15899.918} C_VEL
LIN {X 0,Y 373.597,Z 1123.989,A -85,B 0,C 180,E1 15896.993,E2 15896.993} C_VEL
LIN {X 0,Y 374.75,Z 1120.524,A -85,B 0,C 180,E1 15896.141,E2 15896.141} C_VEL
LIN {X 0,Y 382.501,Z 1105.648,A -85,B 0,C 180,E1 15893.043,E2 15893.043} C_VEL
LIN {X 0,Y 389.805,Z 1091.555,A -85,B 0,C 180,E1 15890.497,E2 15890.497} C_VEL
LIN {X 0,Y 397.757,Z 1075.924,A -85,B 0,C 180,E1 15888.037,E2 15888.037} C_VEL
LIN {X 0,Y 407.798,Z 1055.409,A -85,B 0,C 180,E1 15885.277,E2 15885.277} C_VEL
LIN {X 0,Y 416.511,Z 1036.504,A -85,B 0,C 180,E1 15883.133,E2 15883.133} C_VEL
LIN {X 0,Y 424.077,Z 1019.215,A -85,B 0,C 180,E1 15881.431,E2 15881.431} C_VEL
LIN {X 0,Y 431.379,Z 1001.431,A -85,B 0,C 180,E1 15879.897,E2 15879.897} C_VEL
LIN {X 0,Y 439.855,Z 979.231,A -85,B 0,C 180,E1 15878.245,E2 15878.245} C_VEL
LIN {X 0,Y 448.241,Z 954.508,A -85,B 0,C 180,E1 15876.715,E2 15876.715} C_VEL
LIN {X 0,Y 454.558,Z 933.77,A -85,B 0,C 180,E1 15875.634,E2 15875.634} C_VEL
LIN {X 0,Y 459.973,Z 913.876,A -85,B 0,C 180,E1 15874.748,E2 15874.748} C_VEL
LIN {X 0,Y 464.906,Z 893.261,A -85,B 0,C 180,E1 15873.97,E2 15873.97} C_VEL
LIN {X 0,Y 470.229,Z 867.223,A -85,B 0,C 180,E1 15873.165,E2 15873.165} C_VEL
LIN {X 0,Y 474.431,Z 840.141,A -85,B 0,C 180,E1 15872.534,E2 15872.534} C_VEL
LIN {X 0,Y 476.987,Z 817.634,A -85,B 0,C 180,E1 15872.121,E2 15872.121} C_VEL
LIN {X 0,Y 492.037,Z 611.419,A -85,B 0,C 180,E1 15868.893,E2 15868.893} C_VEL
LIN {X 0,Y 497.306,Z 540.208,A -85,B 0,C 180,E1 15867.776,E2 15867.776} C_VEL
LIN {X 0,Y 488.664,Z 526.43,A -85,B 0,C 180,E1 15864.801,E2 15864.801} C_VEL
LIN {X 0,Y 481.807,Z 516.137,A -85,B 0,C 180,E1 15862.063,E2 15862.063} C_VEL
LIN {X 0,Y 476.506,Z 508.328,A -85,B 0,C 180,E1 15859.586,E2 15859.586} C_VEL
LIN {X 0,Y 472.844,Z 503.077,A -85,B 0,C 180,E1 15857.601,E2 15857.601} C_VEL
LIN {X 0,Y 469.975,Z 498.955,A -85,B 0,C 180,E1 15855.803,E2 15855.803} C_VEL
LIN {X 0,Y 466.831,Z 494.428,A -85,B 0,C 180,E1 15853.438,E2 15853.438} C_VEL
LIN {X 0,Y 463.515,Z 489.948,A -85,B 0,C 180,E1 15850.063,E2 15850.063} C_VEL
LIN {X 0,Y 462.862,Z 488.494,A -85,B 0,C 180,E1 15849.073,E2 15849.073} C_VEL
LIN {X 0,Y 460.932,Z 487.12,A -85,B 0,C 180,E1 15843.773,E2 15843.773} C_VEL
LIN {X 0,Y 462.294,Z 488.187,A -85,B 0,C 180,E1 15838.885,E2 15838.885} C_VEL
LIN {X 0,Y 463.114,Z 488.904,A -85,B 0,C 180,E1 15837.649,E2 15837.649} C_VEL
LIN {X 0,Y 465.227,Z 492.757,A -85,B 0,C 180,E1 15835.068,E2 15835.068} C_VEL
LIN {X 0,Y 466.83,Z 494.419,A -85,B 0,C 180,E1 15833.667,E2 15833.667} C_VEL
LIN {X 0,Y 469.966,Z 498.874,A -85,B 0,C 180,E1 15831.312,E2 15831.312} C_VEL
LIN {X 0,Y 474.378,Z 505.296,A -85,B 0,C 180,E1 15828.634,E2 15828.634} C_VEL
LIN {X 0,Y 478.523,Z 511.299,A -85,B 0,C 180,E1 15826.527,E2 15826.527} C_VEL
LIN {X 0,Y 483.737,Z 518.964,A -85,B 0,C 180,E1 15824.228,E2 15824.228} C_VEL
LIN {X 0,Y 490.555,Z 529.358,A -85,B 0,C 180,E1 15821.613,E2 15821.613} C_VEL
LIN {X 0,Y 497.268,Z 541.146,A -85,B 0,C 180,E1 15819.305,E2 15819.305} C_VEL
LIN {X 0,Y 497.103,Z 544.856,A -85,B 0,C 180,E1 15819.218,E2 15819.218} C_VEL
LIN {X 0,Y 480.932,Z 766.34,A -85,B 0,C 180,E1 15815.769,E2 15815.769} C_VEL
LIN {X 0,Y 476.355,Z 827.145,A -85,B 0,C 180,E1 15814.799,E2 15814.799} C_VEL
LIN {X 0,Y 472.377,Z 857.555,A -85,B 0,C 180,E1 15814.198,E2 15814.198} C_VEL
LIN {X 0,Y 468.307,Z 880.396,A -85,B 0,C 180,E1 15813.611,E2 15813.611} C_VEL
LIN {X 0,Y 463.914,Z 901.158,A -85,B 0,C 180,E1 15812.949,E2 15812.949} C_VEL
LIN {X 0,Y 458.81,Z 921.969,A -85,B 0,C 180,E1 15812.156,E2 15812.156} C_VEL
LIN {X 0,Y 451.851,Z 946.947,A -85,B 0,C 180,E1 15811.012,E2 15811.012} C_VEL
LIN {X 0,Y 443.858,Z 971.554,A -85,B 0,C 180,E1 15809.628,E2 15809.628} C_VEL
LIN {X 0,Y 436.929,Z 990.945,A -85,B 0,C 180,E1 15808.35,E2 15808.35} C_VEL
LIN {X 0,Y 429.642,Z 1009.86,A -85,B 0,C 180,E1 15806.907,E2 15806.907} C_VEL
LIN {X 0,Y 421.637,Z 1029.212,A -85,B 0,C 180,E1 15805.205,E2 15805.205} C_VEL
LIN {X 0,Y 411.208,Z 1052.549,A -85,B 0,C 180,E1 15802.78,E2 15802.78} C_VEL
LIN {X 0,Y 403.154,Z 1069.576,A -85,B 0,C 180,E1 15800.695,E2 15800.695} C_VEL
LIN {X 0,Y 395.551,Z 1085.062,A -85,B 0,C 180,E1 15798.525,E2 15798.525} C_VEL
LIN {X 0,Y 387.935,Z 1100.171,A -85,B 0,C 180,E1 15796.105,E2 15796.105} C_VEL
LIN {X 0,Y 379.077,Z 1117.514,A -85,B 0,C 180,E1 15792.883,E2 15792.883} C_VEL
LIN {X 0,Y 371.443,Z 1132.178,A -85,B 0,C 180,E1 15789.64,E2 15789.64} C_VEL
LIN {X 0,Y 365.434,Z 1144.009,A -85,B 0,C 180,E1 15786.617,E2 15786.617} C_VEL
LIN {X 0,Y 360.264,Z 1154.554,A -85,B 0,C 180,E1 15783.524,E2 15783.524} C_VEL
LIN {X 0,Y 355.314,Z 1165.203,A -85,B 0,C 180,E1 15779.917,E2 15779.917} C_VEL
LIN {X 0,Y 350.552,Z 1176.525,A -85,B 0,C 180,E1 15775.285,E2 15775.285} C_VEL
LIN {X 0,Y 347.839,Z 1183.95,A -85,B 0,C 180,E1 15771.588,E2 15771.588} C_VEL
LIN {X 0,Y 346.035,Z 1189.845,A -85,B 0,C 180,E1 15768.071,E2 15768.071} C_VEL
LIN {X 0,Y 344.912,Z 1194.596,A -85,B 0,C 180,E1 15764.608,E2 15764.608} C_VEL
LIN {X 0,Y 344.256,Z 1198.428,A -85,B 0,C 180,E1 15761.051,E2 15761.051} C_VEL
LIN {X 0,Y 343.999,Z 1201.204,A -85,B 0,C 180,E1 15757.516,E2 15757.516} C_VEL
LIN {X 0,Y 343.915,Z 1203.084,A -85,B 0,C 180,E1 15753.667,E2 15753.667} C_VEL
LIN {X 0,Y 343.913,Z 1203.756,A -85,B 0,C 180,E1 15749.667,E2 15749.667} C_VEL
LIN {X 0,Y 343.918,Z 1202.994,A -85,B 0,C 180,E1 15745.665,E2 15745.665} C_VEL
LIN {X 0,Y 344.016,Z 1201.183,A -85,B 0,C 180,E1 15741.981,E2 15741.981} C_VEL
LIN {X 0,Y 344.325,Z 1198.435,A -85,B 0,C 180,E1 15738.442,E2 15738.442} C_VEL
LIN {X 0,Y 345.068,Z 1194.669,A -85,B 0,C 180,E1 15734.884,E2 15734.884} C_VEL
LIN {X 0,Y 346.392,Z 1189.738,A -85,B 0,C 180,E1 15731.228,E2 15731.228} C_VEL
LIN {X 0,Y 348.361,Z 1183.989,A -85,B 0,C 180,E1 15727.737,E2 15727.737} C_VEL
LIN {X 0,Y 351.34,Z 1176.66,A -85,B 0,C 180,E1 15724.007,E2 15724.007} C_VEL
LIN {X 0,Y 356.379,Z 1165.918,A -85,B 0,C 180,E1 15719.469,E2 15719.469} C_VEL
LIN {X 0,Y 361.927,Z 1155.085,A -85,B 0,C 180,E1 15715.695,E2 15715.695} C_VEL
LIN {X 0,Y 367.749,Z 1144.379,A -85,B 0,C 180,E1 15712.481,E2 15712.481} C_VEL
LIN {X 0,Y 374.549,Z 1132.354,A -85,B 0,C 180,E1 15709.356,E2 15709.356} C_VEL
LIN {X 0,Y 383.529,Z 1116.827,A -85,B 0,C 180,E1 15705.888,E2 15705.888} C_VEL
LIN {X 0,Y 393.183,Z 1099.69,A -85,B 0,C 180,E1 15702.7,E2 15702.7} C_VEL
LIN {X 0,Y 401.405,Z 1084.964,A -85,B 0,C 180,E1 15700.34,E2 15700.34} C_VEL
LIN {X 0,Y 409.713,Z 1069.678,A -85,B 0,C 180,E1 15698.205,E2 15698.205} C_VEL
LIN {X 0,Y 417.974,Z 1053.898,A -85,B 0,C 180,E1 15696.278,E2 15696.278} C_VEL
LIN {X 0,Y 428.181,Z 1033.487,A -85,B 0,C 180,E1 15694.127,E2 15694.127} C_VEL
LIN {X 0,Y 438.296,Z 1011.458,A -85,B 0,C 180,E1 15692.185,E2 15692.185} C_VEL
LIN {X 0,Y 446.27,Z 992.755,A -85,B 0,C 180,E1 15690.771,E2 15690.771} C_VEL
LIN {X 0,Y 453.853,Z 973.538,A -85,B 0,C 180,E1 15689.518,E2 15689.518} C_VEL
LIN {X 0,Y 460.97,Z 953.826,A -85,B 0,C 180,E1 15688.413,E2 15688.413} C_VEL
LIN {X 0,Y 468.62,Z 930.293,A -85,B 0,C 180,E1 15687.296,E2 15687.296} C_VEL
LIN {X 0,Y 475.881,Z 904.026,A -85,B 0,C 180,E1 15686.288,E2 15686.288} C_VEL
LIN {X 0,Y 481.067,Z 881.935,A -85,B 0,C 180,E1 15685.601,E2 15685.601} C_VEL
LIN {X 0,Y 485.246,Z 860.817,A -85,B 0,C 180,E1 15685.07,E2 15685.07} C_VEL
LIN {X 0,Y 488.867,Z 837.961,A -85,B 0,C 180,E1 15684.608,E2 15684.608} C_VEL
LIN {X 0,Y 492.259,Z 805.464,A -85,B 0,C 180,E1 15684.063,E2 15684.063} C_VEL
LIN {X 0,Y 510.58,Z 584.491,A -85,B 0,C 180,E1 15680.651,E2 15680.651} C_VEL
LIN {X 0,Y 513.499,Z 549.918,A -85,B 0,C 180,E1 15680.102,E2 15680.102} C_VEL
LIN {X 0,Y 510.005,Z 543.77,A -85,B 0,C 180,E1 15678.459,E2 15678.459} C_VEL
LIN {X 0,Y 505.752,Z 536.938,A -85,B 0,C 180,E1 15676.186,E2 15676.186} C_VEL
LIN {X 0,Y 502.486,Z 531.93,A -85,B 0,C 180,E1 15674.109,E2 15674.109} C_VEL
LIN {X 0,Y 499.673,Z 527.613,A -85,B 0,C 180,E1 15671.895,E2 15671.895} C_VEL
LIN {X 0,Y 496.805,Z 522.868,A -85,B 0,C 180,E1 15668.682,E2 15668.682} C_VEL
LIN {X 0,Y 494.896,Z 520.949,A -85,B 0,C 180,E1 15663.823,E2 15663.823} C_VEL
LIN {X 0,Y 495.287,Z 521.543,A -85,B 0,C 180,E1 15660.925,E2 15660.925} C_VEL
LIN {X 0,Y 497.025,Z 523.174,A -85,B 0,C 180,E1 15657.809,E2 15657.809} C_VEL
LIN {X 0,Y 499.749,Z 527.7,A -85,B 0,C 180,E1 15654.834,E2 15654.834} C_VEL
LIN {X 0,Y 503.572,Z 533.545,A -85,B 0,C 180,E1 15651.953,E2 15651.953} C_VEL
LIN {X 0,Y 507.105,Z 539.166,A -85,B 0,C 180,E1 15649.836,E2 15649.836} C_VEL
LIN {X 0,Y 511.593,Z 546.157,A -85,B 0,C 180,E1 15647.585,E2 15647.585} C_VEL
LIN {X 0,Y 513.486,Z 549.455,A -85,B 0,C 180,E1 15646.72,E2 15646.72} C_VEL
LIN {X 0,Y 495.504,Z 763.839,A -85,B 0,C 180,E1 15643.415,E2 15643.415} C_VEL
LIN {X 0,Y 490.434,Z 822.826,A -85,B 0,C 180,E1 15642.485,E2 15642.485} C_VEL
LIN {X 0,Y 486.166,Z 852.839,A -85,B 0,C 180,E1 15641.907,E2 15641.907} C_VEL
LIN {X 0,Y 481.814,Z 875.526,A -85,B 0,C 180,E1 15641.339,E2 15641.339} C_VEL
LIN {X 0,Y 477.018,Z 896.442,A -85,B 0,C 180,E1 15640.691,E2 15640.691} C_VEL
LIN {X 0,Y 471.572,Z 916.918,A -85,B 0,C 180,E1 15639.93,E2 15639.93} C_VEL
LIN {X 0,Y 464.611,Z 939.911,A -85,B 0,C 180,E1 15638.909,E2 15638.909} C_VEL
LIN {X 0,Y 455.571,Z 965.692,A -85,B 0,C 180,E1 15637.515,E2 15637.515} C_VEL
LIN {X 0,Y 447.879,Z 985.375,A -85,B 0,C 180,E1 15636.247,E2 15636.247} C_VEL
LIN {X 0,Y 439.981,Z 1004.031,A -85,B 0,C 180,E1 15634.851,E2 15634.851} C_VEL
LIN {X 0,Y 431.787,Z 1022.006,A -85,B 0,C 180,E1 15633.304,E2 15633.304} C_VEL
LIN {X 0,Y 421.289,Z 1043.623,A -85,B 0,C 180,E1 15631.135,E2 15631.135} C_VEL
LIN {X 0,Y 411.037,Z 1063.09,A -85,B 0,C 180,E1 15628.792,E2 15628.792} C_VEL
LIN {X 0,Y 402.698,Z 1078.332,A -85,B 0,C 180,E1 15626.667,E2 15626.667} C_VEL
LIN {X 0,Y 394.47,Z 1092.909,A -85,B 0,C 180,E1 15624.338,E2 15624.338} C_VEL
LIN {X 0,Y 386.16,Z 1107.369,A -85,B 0,C 180,E1 15621.678,E2 15621.678} C_VEL
LIN {X 0,Y 376.039,Z 1124.771,A -85,B 0,C 180,E1 15617.888,E2 15617.888} C_VEL
LIN {X 0,Y 368.726,Z 1137.382,A -85,B 0,C 180,E1 15614.613,E2 15614.613} C_VEL
LIN {X 0,Y 362.785,Z 1148.009,A -85,B 0,C 180,E1 15611.411,E2 15611.411} C_VEL
LIN {X 0,Y 357.287,Z 1158.341,A -85,B 0,C 180,E1 15607.797,E2 15607.797} C_VEL
LIN {X 0,Y 351.784,Z 1169.626,A -85,B 0,C 180,E1 15603.018,E2 15603.018} C_VEL
LIN {X 0,Y 348.614,Z 1177.034,A -85,B 0,C 180,E1 15599.181,E2 15599.181} C_VEL
